REGION Network 7: ET01 >>> Lectura de CARA DELANTERA
   RUNG wire#powerrail
      Contact( #GAL_ET00 )
      Contact( #HabilitarLectura )
      Contact( #PermisoLectura )
      Contact( #pHsGalibo_OK )
      Contact( #pHs_LecturaDelantera_Des1 )
      Contact( #pHs_LecturaTrasera_Des1 )
      Contact( #pHs_LecturaDelantera_Des2 )
      Contact( #pHs_LecturaTrasera_Des2 )
      Contact( #pHs_LecturaDelantera_Error )
      Contact( #pHs_LecturaTrasera_Error )
      Contact( #EstadoZona.Marcha_CBx )
      I_Contact( #EstadoZona.Error_CBx )
      S_SR(operand := #GAL_ET01, r1 := wire#w1)
   END_RUNG
   RUNG wire#powerrail
      Contact( #GAL_ET02 )
   END_RUNG wire#w1
   RUNG wire#powerrail
      Contact( #EstadoZona.Resetear_CBx )
   END_RUNG wire#w1
   // the same network as SCL:
   IF #GAL_ET00 AND #HabilitarLectura AND #PermisoLectura AND #pHsGalibo_OK AND #pHs_LecturaDelantera_Des1 AND #pHs_LecturaTrasera_Des1 AND #pHs_LecturaDelantera_Des2 AND #pHs_LecturaTrasera_Des2 AND #pHs_LecturaDelantera_Error AND #pHs_LecturaTrasera_Error AND #EstadoZona.Marcha_CBx AND NOT #EstadoZona.Error_CBx THEN
       #GAL_ET01 := TRUE;   // SR flip-flop
   END_IF;
   IF #GAL_ET02 OR #EstadoZona.Resetear_CBx THEN #GAL_ET01 := FALSE; END_IF;
END_REGION

REGION Network 8: ET00 >>> INICIO
   RUNG wire#powerrail
      I_Contact( #GAL_ET00 )
      I_Contact( #GAL_ET01 )
      I_Contact( #GAL_ET02 )
      I_Contact( #GAL_ET03 )
      I_Contact( #GAL_ET04 )
      wire#w1
      S_SR(operand := #GAL_ET00, r1 := wire#w2)
   END_RUNG
   RUNG wire#powerrail
      Contact( #GAL_ET04 )
      I_Contact( #HabilitarLectura )
      I_Contact( #PermisoLectura )
      Contact( #pHsGalibo_OK )
      Contact( #pHs_LecturaDelantera_Des1 )
      Contact( #pHs_LecturaTrasera_Des1 )
      Contact( #pHs_LecturaDelantera_Des2 )
      Contact( #pHs_LecturaTrasera_Des2 )
      Contact( #pHs_LecturaDelantera_Error )
      Contact( #pHs_LecturaTrasera_Error )
   END_RUNG wire#w1
   RUNG wire#powerrail
      Contact( #GAL_ET01 )
   END_RUNG wire#w2
   RUNG wire#powerrail
      Contact( #EstadoZona.Resetear_CBx )
   END_RUNG wire#w2
   // the same network as SCL:
   IF (NOT #GAL_ET00 AND NOT #GAL_ET01 AND NOT #GAL_ET02 AND NOT #GAL_ET03 AND NOT #GAL_ET04) OR (#GAL_ET04 AND NOT #HabilitarLectura AND NOT #PermisoLectura AND #pHsGalibo_OK AND #pHs_LecturaDelantera_Des1 AND #pHs_LecturaTrasera_Des1 AND #pHs_LecturaDelantera_Des2 AND #pHs_LecturaTrasera_Des2 AND #pHs_LecturaDelantera_Error AND #pHs_LecturaTrasera_Error) THEN
       #GAL_ET00 := TRUE;   // SR flip-flop
   END_IF;
   IF #GAL_ET01 OR #EstadoZona.Resetear_CBx THEN #GAL_ET00 := FALSE; END_IF;
END_REGION

REGION Network 9: ERROR >>> Fotocelulas de Galibo
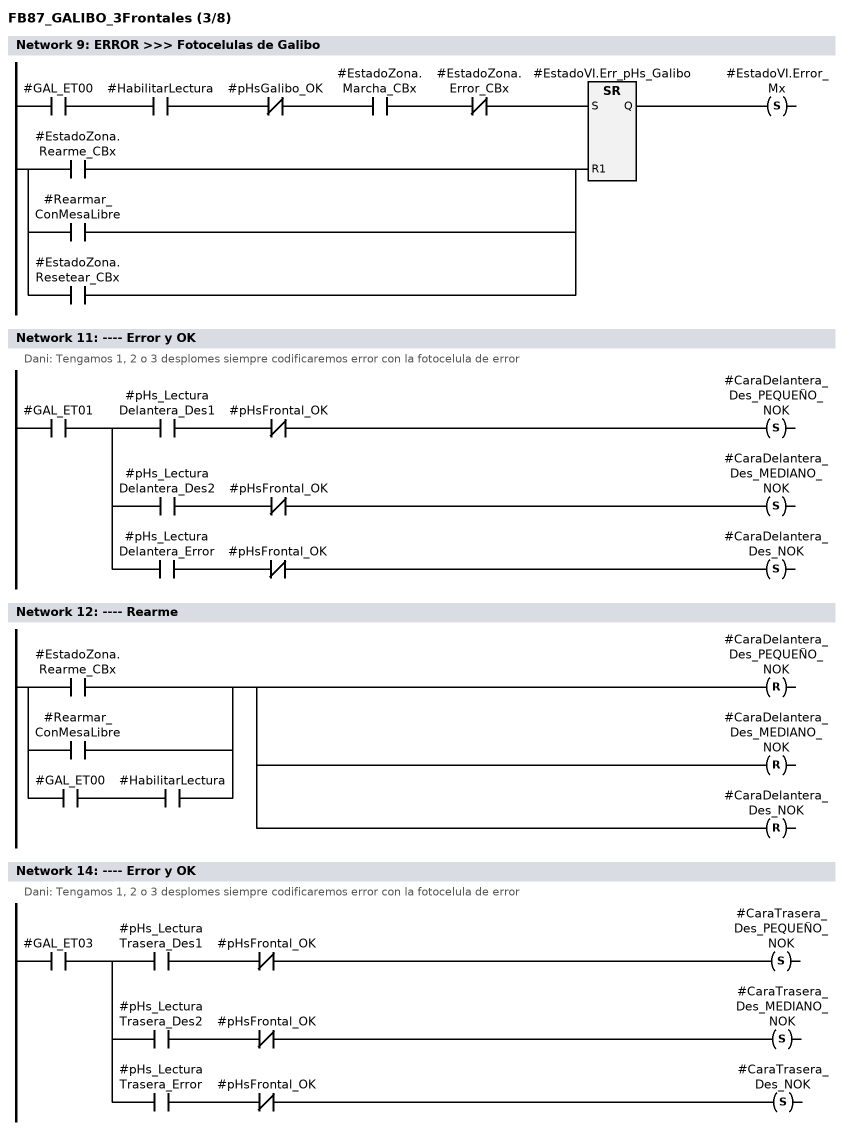
   RUNG wire#powerrail
      Contact( #GAL_ET00 )
      Contact( #HabilitarLectura )
      I_Contact( #pHsGalibo_OK )
      Contact( #EstadoZona.Marcha_CBx )
      I_Contact( #EstadoZona.Error_CBx )
      S_SR(operand := #EstadoVI.Err_pHs_Galibo, r1 := wire#w1)
      S_Coil( #EstadoVI.Error_Mx )
   END_RUNG
   RUNG wire#powerrail
      Contact( #EstadoZona.Rearme_CBx )
   END_RUNG wire#w1
   RUNG wire#powerrail
      Contact( #Rearmar_ConMesaLibre )
   END_RUNG wire#w1
   RUNG wire#powerrail
      Contact( #EstadoZona.Resetear_CBx )
   END_RUNG wire#w1
   // the same network as SCL:
   IF #GAL_ET00 AND #HabilitarLectura AND NOT #pHsGalibo_OK AND #EstadoZona.Marcha_CBx AND NOT #EstadoZona.Error_CBx THEN
       #EstadoVI.Err_pHs_Galibo := TRUE;   // SR flip-flop
   END_IF;
   IF #EstadoZona.Rearme_CBx OR #Rearmar_ConMesaLibre OR #EstadoZona.Resetear_CBx THEN
       #EstadoVI.Err_pHs_Galibo := FALSE;
   END_IF;
   IF #EstadoVI.Err_pHs_Galibo THEN #EstadoVI.Error_Mx := TRUE; END_IF;
END_REGION

REGION Network 10: VARIABLES DE CONTROL DE LARGURA >>> Activar la lectura de Cara Delantera
END_REGION

REGION Network 11: ---- Error y OK
   // Dani: Tengamos 1, 2 o 3 desplomes siempre codificaremos error con la fotocelula de error
   RUNG wire#powerrail
      Contact( #GAL_ET01 )
      wire#w1
      Contact( #pHs_LecturaDelantera_Des1 )
      I_Contact( #pHsFrontal_OK )
      S_Coil( #CaraDelantera_Des_PEQUEÑO_NOK )
   END_RUNG
   RUNG wire#w1
      Contact( #pHs_LecturaDelantera_Des2 )
      I_Contact( #pHsFrontal_OK )
      S_Coil( #CaraDelantera_Des_MEDIANO_NOK )
   END_RUNG
   RUNG wire#w1
      Contact( #pHs_LecturaDelantera_Error )
      I_Contact( #pHsFrontal_OK )
      S_Coil( #CaraDelantera_Des_NOK )
   END_RUNG
   // the same network as SCL:
   IF #GAL_ET01 AND #pHs_LecturaDelantera_Des1 AND NOT #pHsFrontal_OK THEN
       #CaraDelantera_Des_PEQUEÑO_NOK := TRUE;
   END_IF;
   IF #GAL_ET01 AND #pHs_LecturaDelantera_Des2 AND NOT #pHsFrontal_OK THEN
       #CaraDelantera_Des_MEDIANO_NOK := TRUE;
   END_IF;
   IF #GAL_ET01 AND #pHs_LecturaDelantera_Error AND NOT #pHsFrontal_OK THEN
       #CaraDelantera_Des_NOK := TRUE;
   END_IF;
END_REGION

REGION Network 12: ---- Rearme
   RUNG wire#powerrail
      Contact( #EstadoZona.Rearme_CBx )
      wire#w1
      R_Coil( #CaraDelantera_Des_PEQUEÑO_NOK )
   END_RUNG
   RUNG wire#powerrail
      Contact( #Rearmar_ConMesaLibre )
   END_RUNG wire#w1
   RUNG wire#powerrail
      Contact( #GAL_ET00 )
      Contact( #HabilitarLectura )
   END_RUNG wire#w1
   RUNG wire#w1
      R_Coil( #CaraDelantera_Des_MEDIANO_NOK )
   END_RUNG
   RUNG wire#w1
      R_Coil( #CaraDelantera_Des_NOK )
   END_RUNG
   // the same network as SCL:
   IF #EstadoZona.Rearme_CBx OR #Rearmar_ConMesaLibre OR (#GAL_ET00 AND #HabilitarLectura) THEN
       #CaraDelantera_Des_PEQUEÑO_NOK := FALSE;
       #CaraDelantera_Des_MEDIANO_NOK := FALSE;
       #CaraDelantera_Des_NOK := FALSE;
   END_IF;
END_REGION

REGION Network 13: VARIABLES DE CONTROL DE LARGURA >>> Activar la lectura de Cara Trasera
END_REGION

REGION Network 14: ---- Error y OK
   // Dani: Tengamos 1, 2 o 3 desplomes siempre codificaremos error con la fotocelula de error
   RUNG wire#powerrail
      Contact( #GAL_ET03 )
      wire#w1
      Contact( #pHs_LecturaTrasera_Des1 )
      I_Contact( #pHsFrontal_OK )
      S_Coil( #CaraTrasera_Des_PEQUEÑO_NOK )
   END_RUNG
   RUNG wire#w1
      Contact( #pHs_LecturaTrasera_Des2 )
      I_Contact( #pHsFrontal_OK )
      S_Coil( #CaraTrasera_Des_MEDIANO_NOK )
   END_RUNG
   RUNG wire#w1
      Contact( #pHs_LecturaTrasera_Error )
      I_Contact( #pHsFrontal_OK )
      S_Coil( #CaraTrasera_Des_NOK )
   END_RUNG
   // the same network as SCL:
   IF #GAL_ET03 AND #pHs_LecturaTrasera_Des1 AND NOT #pHsFrontal_OK THEN
       #CaraTrasera_Des_PEQUEÑO_NOK := TRUE;
   END_IF;
   IF #GAL_ET03 AND #pHs_LecturaTrasera_Des2 AND NOT #pHsFrontal_OK THEN
       #CaraTrasera_Des_MEDIANO_NOK := TRUE;
   END_IF;
   IF #GAL_ET03 AND #pHs_LecturaTrasera_Error AND NOT #pHsFrontal_OK THEN
       #CaraTrasera_Des_NOK := TRUE;
   END_IF;
END_REGION

REGION Network 15: ---- Rearme
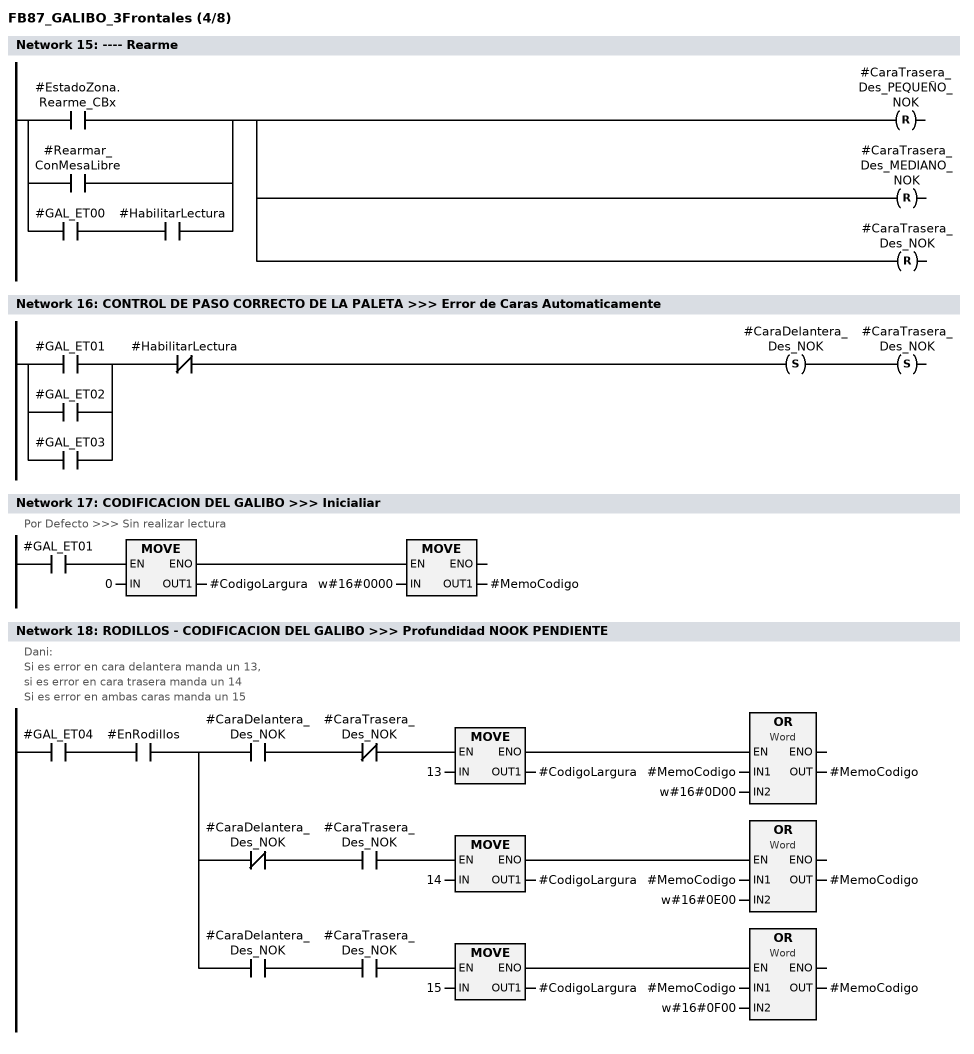
   RUNG wire#powerrail
      Contact( #EstadoZona.Rearme_CBx )
      wire#w1
      R_Coil( #CaraTrasera_Des_PEQUEÑO_NOK )
   END_RUNG
   RUNG wire#powerrail
      Contact( #Rearmar_ConMesaLibre )
   END_RUNG wire#w1
   RUNG wire#powerrail
      Contact( #GAL_ET00 )
      Contact( #HabilitarLectura )
   END_RUNG wire#w1
   RUNG wire#w1
      R_Coil( #CaraTrasera_Des_MEDIANO_NOK )
   END_RUNG
   RUNG wire#w1
      R_Coil( #CaraTrasera_Des_NOK )
   END_RUNG
   // the same network as SCL:
   IF #EstadoZona.Rearme_CBx OR #Rearmar_ConMesaLibre OR (#GAL_ET00 AND #HabilitarLectura) THEN
       #CaraTrasera_Des_PEQUEÑO_NOK := FALSE;
       #CaraTrasera_Des_MEDIANO_NOK := FALSE;
       #CaraTrasera_Des_NOK := FALSE;
   END_IF;
END_REGION

REGION Network 16: CONTROL DE PASO CORRECTO DE LA PALETA >>> Error de Caras Automaticamente
   RUNG wire#powerrail
      Contact( #GAL_ET01 )
      wire#w1
      I_Contact( #HabilitarLectura )
      S_Coil( #CaraDelantera_Des_NOK )
      S_Coil( #CaraTrasera_Des_NOK )
   END_RUNG
   RUNG wire#powerrail
      Contact( #GAL_ET02 )
   END_RUNG wire#w1
   RUNG wire#powerrail
      Contact( #GAL_ET03 )
   END_RUNG wire#w1
   // the same network as SCL:
   IF (#GAL_ET01 OR #GAL_ET02 OR #GAL_ET03) AND NOT #HabilitarLectura THEN
       #CaraDelantera_Des_NOK := TRUE;
       #CaraTrasera_Des_NOK := TRUE;
   END_IF;
END_REGION

REGION Network 17: CODIFICACION DEL GALIBO >>> Inicialiar
   // Por Defecto >>> Sin realizar lectura
   RUNG wire#powerrail
      Contact( #GAL_ET01 )
      { S7_GenerateENO := "TRUE" } Move(in := 0, out1 => #CodigoLargura)
      { S7_GenerateENO := "TRUE" } Move(in := w#16#0000, out1 => #MemoCodigo)
   END_RUNG
   // the same network as SCL:
   // ENO of a box is taken as its EN; it also drops when the box reports an error
   IF #GAL_ET01 THEN
       #CodigoLargura := 0;
       #MemoCodigo := w#16#0000;
   END_IF;
END_REGION

REGION Network 18: RODILLOS - CODIFICACION DEL GALIBO >>> Profundidad NOOK PENDIENTE
   // Dani:
   // Si es error en cara delantera manda un 13, 
   // si es error en cara trasera manda un 14
   // Si es error en ambas caras manda un 15
   #_w1 := #GAL_ET04 AND #EnRodillos;
   IF #_w1 AND #CaraDelantera_Des_NOK AND NOT #CaraTrasera_Des_NOK THEN
       #CodigoLargura := 13;
       #MemoCodigo := #MemoCodigo OR w#16#0D00;
   END_IF;
   IF #_w1 AND NOT #CaraDelantera_Des_NOK AND #CaraTrasera_Des_NOK THEN
       #CodigoLargura := 14;
       #MemoCodigo := #MemoCodigo OR w#16#0E00;
   END_IF;
   IF #_w1 AND #CaraDelantera_Des_NOK AND #CaraTrasera_Des_NOK THEN
       #CodigoLargura := 15;
       #MemoCodigo := #MemoCodigo OR w#16#0F00;
   END_IF;
END_REGION

REGION Network 19: RODILLOS - CODIFICACION DEL GALIBO >>> Profundidad OK - Codificacion
   // Dani:  los Nook solo se escriben si el desplome esta configurado
   // si hay 1 desplome envia 1 si la carga no da error de desplome
   // Si hay 2 desplomes envia 1 si no hay desplome pequeño y 2 si no hay error de desplome
   // Si hay 3 desplomes envia 1 si no hay desplome pequeño, 2 si no hay desplome mediano y 3 si no hay error de desplome
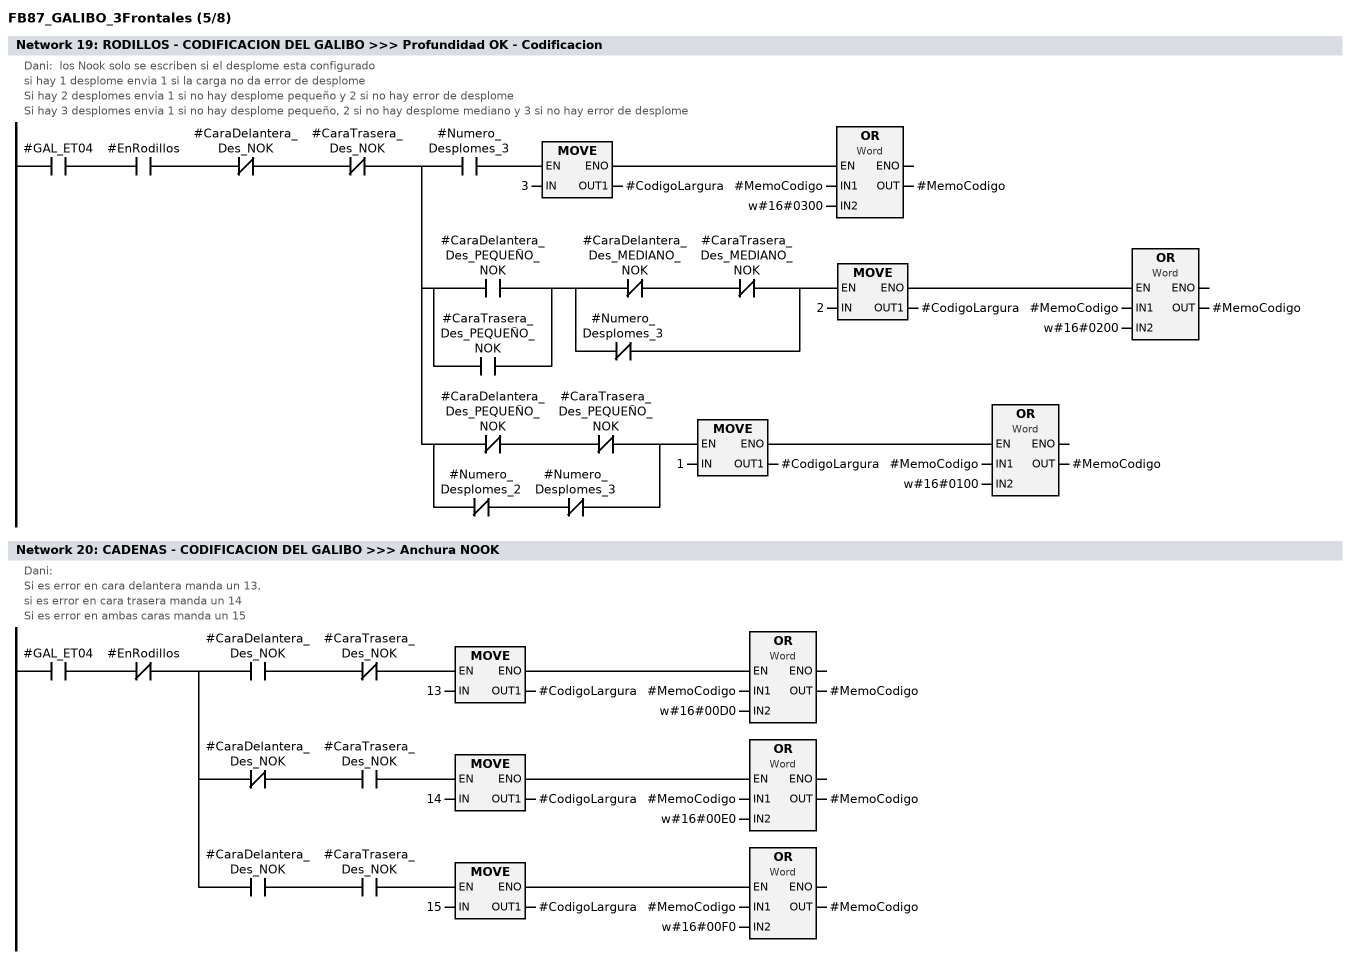
   #_w1 := #GAL_ET04 AND #EnRodillos AND NOT #CaraDelantera_Des_NOK AND NOT #CaraTrasera_Des_NOK;
   IF #_w1 AND #Numero_Desplomes_3 THEN
       #CodigoLargura := 3;
       #MemoCodigo := #MemoCodigo OR w#16#0300;
   END_IF;
   IF #_w1 AND (#CaraDelantera_Des_PEQUEÑO_NOK OR #CaraTrasera_Des_PEQUEÑO_NOK) AND ((NOT #CaraDelantera_Des_MEDIANO_NOK AND NOT #CaraTrasera_Des_MEDIANO_NOK) OR NOT #Numero_Desplomes_3) THEN
       #CodigoLargura := 2;
       #MemoCodigo := #MemoCodigo OR w#16#0200;
   END_IF;
   IF #_w1 AND ((NOT #CaraDelantera_Des_PEQUEÑO_NOK AND NOT #CaraTrasera_Des_PEQUEÑO_NOK) OR (NOT #Numero_Desplomes_2 AND NOT #Numero_Desplomes_3)) THEN
       #CodigoLargura := 1;
       #MemoCodigo := #MemoCodigo OR w#16#0100;
   END_IF;
END_REGION

REGION Network 20: CADENAS - CODIFICACION DEL GALIBO >>> Anchura NOOK
   // Dani:
   // Si es error en cara delantera manda un 13, 
   // si es error en cara trasera manda un 14
   // Si es error en ambas caras manda un 15
   #_w1 := #GAL_ET04 AND NOT #EnRodillos;
   IF #_w1 AND #CaraDelantera_Des_NOK AND NOT #CaraTrasera_Des_NOK THEN
       #CodigoLargura := 13;
       #MemoCodigo := #MemoCodigo OR w#16#00D0;
   END_IF;
   IF #_w1 AND NOT #CaraDelantera_Des_NOK AND #CaraTrasera_Des_NOK THEN
       #CodigoLargura := 14;
       #MemoCodigo := #MemoCodigo OR w#16#00E0;
   END_IF;
   IF #_w1 AND #CaraDelantera_Des_NOK AND #CaraTrasera_Des_NOK THEN
       #CodigoLargura := 15;
       #MemoCodigo := #MemoCodigo OR w#16#00F0;
   END_IF;
END_REGION

REGION Network 21: CADENAS - CODIFICACION DEL GALIBO >>> Anchura OK - Codificacion
   // Dani:
   // Si la cargaes menor que desplome 1 manda 1
   // si la carga es mayor que desplome 1 y menor que desplome 2 manda 2
   // si la carga es mayor que desplome 2 y menor que desplome 3 manda 3
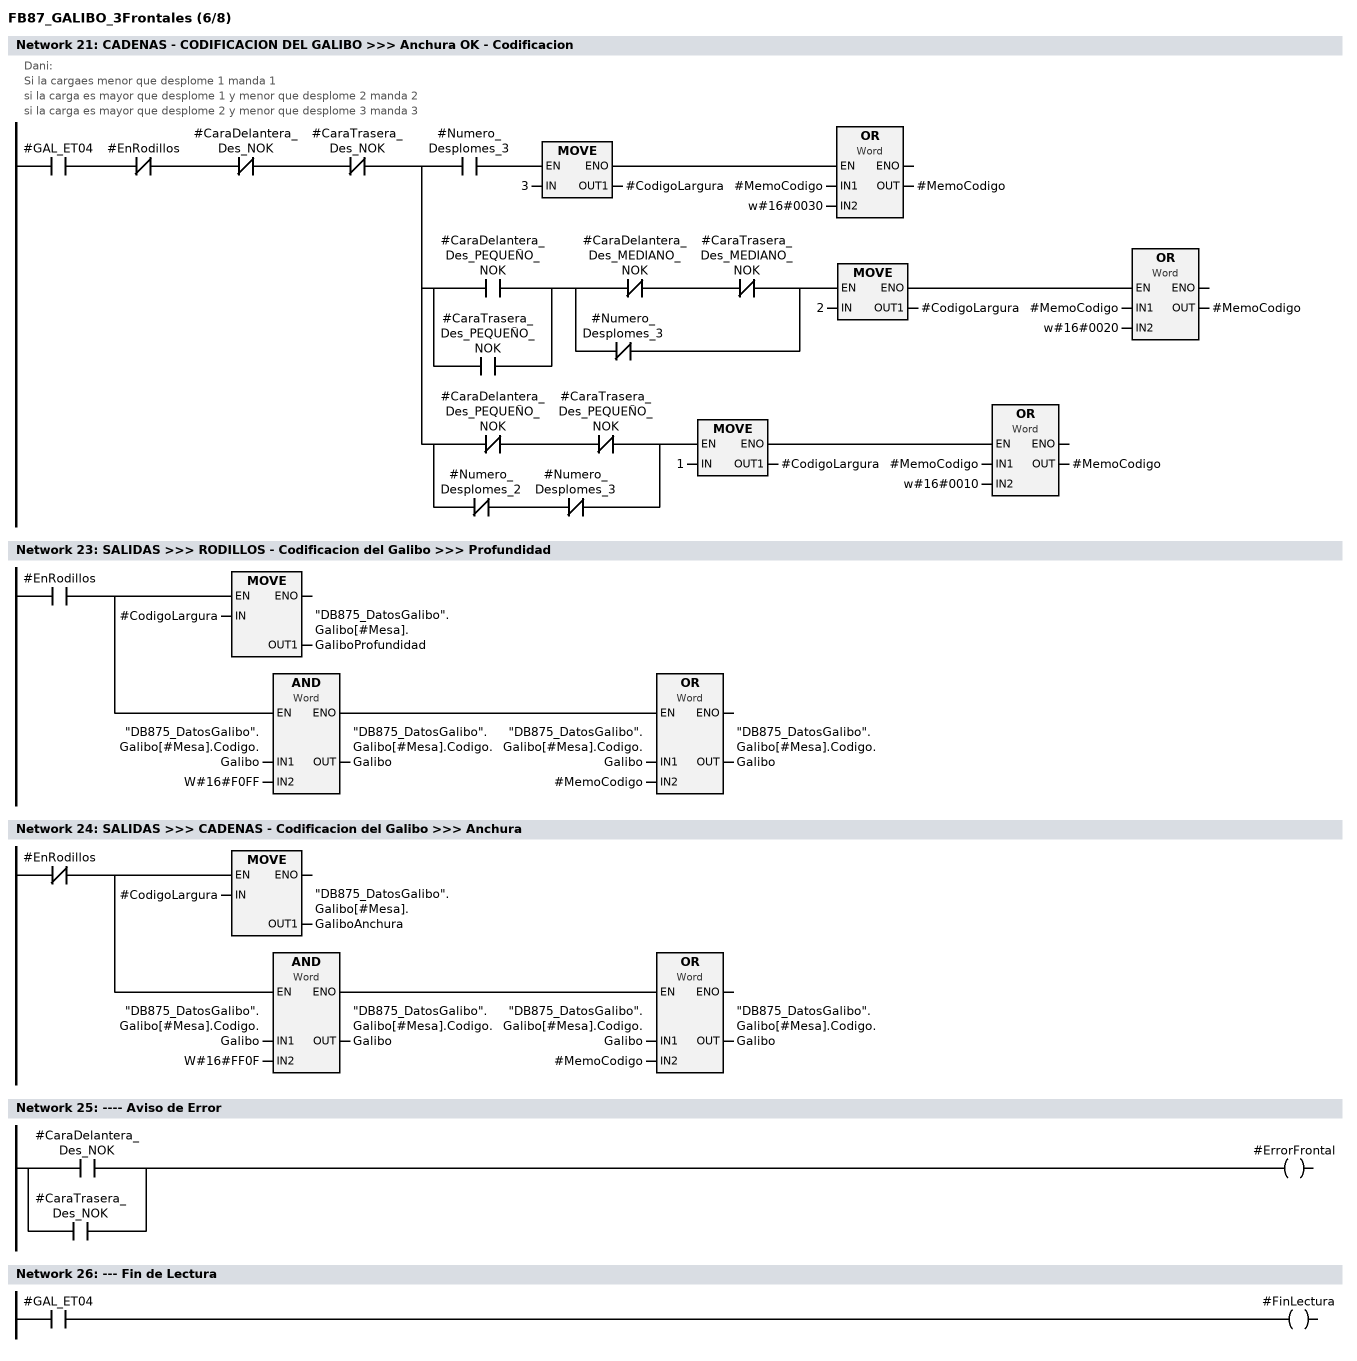
   #_w1 := #GAL_ET04 AND NOT #EnRodillos AND NOT #CaraDelantera_Des_NOK AND NOT #CaraTrasera_Des_NOK;
   IF #_w1 AND #Numero_Desplomes_3 THEN
       #CodigoLargura := 3;
       #MemoCodigo := #MemoCodigo OR w#16#0030;
   END_IF;
   IF #_w1 AND (#CaraDelantera_Des_PEQUEÑO_NOK OR #CaraTrasera_Des_PEQUEÑO_NOK) AND ((NOT #CaraDelantera_Des_MEDIANO_NOK AND NOT #CaraTrasera_Des_MEDIANO_NOK) OR NOT #Numero_Desplomes_3) THEN
       #CodigoLargura := 2;
       #MemoCodigo := #MemoCodigo OR w#16#0020;
   END_IF;
   IF #_w1 AND ((NOT #CaraDelantera_Des_PEQUEÑO_NOK AND NOT #CaraTrasera_Des_PEQUEÑO_NOK) OR (NOT #Numero_Desplomes_2 AND NOT #Numero_Desplomes_3)) THEN
       #CodigoLargura := 1;
       #MemoCodigo := #MemoCodigo OR w#16#0010;
   END_IF;
END_REGION

REGION Network 22: SALIDAS >>> Codificacion del Galibo y Error de Anchura
END_REGION

REGION Network 23: SALIDAS >>> RODILLOS - Codificacion del Galibo >>> Profundidad
   IF #EnRodillos THEN
       "DB875_DatosGalibo".Galibo[#Mesa].GaliboProfundidad := #CodigoLargura;
       "DB875_DatosGalibo".Galibo[#Mesa].Codigo.Galibo := "DB875_DatosGalibo".Galibo[#Mesa].Codigo.Galibo AND W#16#F0FF;
       "DB875_DatosGalibo".Galibo[#Mesa].Codigo.Galibo := "DB875_DatosGalibo".Galibo[#Mesa].Codigo.Galibo OR #MemoCodigo;
   END_IF;
END_REGION

REGION Network 24: SALIDAS >>> CADENAS - Codificacion del Galibo >>> Anchura
   IF NOT #EnRodillos THEN
       "DB875_DatosGalibo".Galibo[#Mesa].GaliboAnchura := #CodigoLargura;
       "DB875_DatosGalibo".Galibo[#Mesa].Codigo.Galibo := "DB875_DatosGalibo".Galibo[#Mesa].Codigo.Galibo AND W#16#FF0F;
       "DB875_DatosGalibo".Galibo[#Mesa].Codigo.Galibo := "DB875_DatosGalibo".Galibo[#Mesa].Codigo.Galibo OR #MemoCodigo;
   END_IF;
END_REGION

REGION Network 25: ---- Aviso de Error
   RUNG wire#powerrail
      Contact( #CaraDelantera_Des_NOK )
      wire#w1
      Coil( #ErrorFrontal )
   END_RUNG
   RUNG wire#powerrail
      Contact( #CaraTrasera_Des_NOK )
   END_RUNG wire#w1
   // the same network as SCL:
   #ErrorFrontal := #CaraDelantera_Des_NOK OR #CaraTrasera_Des_NOK;
END_REGION

REGION Network 26: --- Fin de Lectura
   RUNG wire#powerrail
      Contact( #GAL_ET04 )
      Coil( #FinLectura )
   END_RUNG
   // the same network as SCL:
   #FinLectura := #GAL_ET04;
END_REGION

REGION Network 27: SALIDAS >>> BALIZA
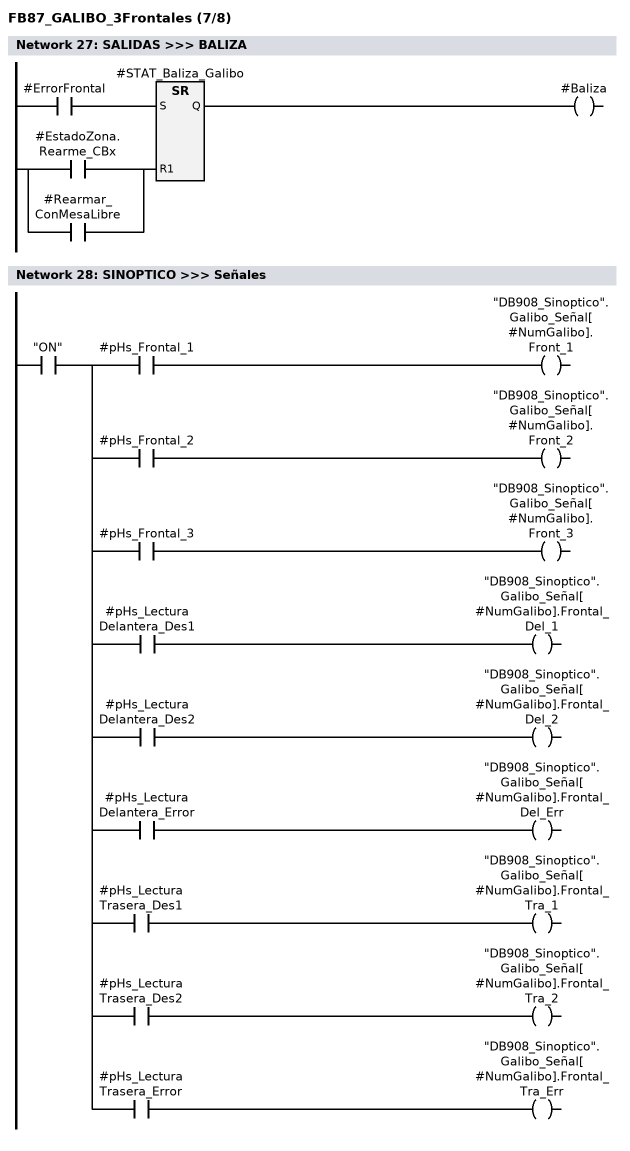
   RUNG wire#powerrail
      Contact( #ErrorFrontal )
      S_SR(operand := #STAT_Baliza_Galibo, r1 := wire#w1)
      Coil( #Baliza )
   END_RUNG
   RUNG wire#powerrail
      Contact( #EstadoZona.Rearme_CBx )
   END_RUNG wire#w1
   RUNG wire#powerrail
      Contact( #Rearmar_ConMesaLibre )
   END_RUNG wire#w1
   // the same network as SCL:
   IF #ErrorFrontal THEN
       #STAT_Baliza_Galibo := TRUE;   // SR flip-flop
   END_IF;
   IF #EstadoZona.Rearme_CBx OR #Rearmar_ConMesaLibre THEN #STAT_Baliza_Galibo := FALSE; END_IF;
   #Baliza := #STAT_Baliza_Galibo;
END_REGION

REGION Network 28: SINOPTICO >>> Señales
   RUNG wire#powerrail
      Contact( "ON" )
      wire#w1
      Contact( #pHs_Frontal_1 )
      Coil( "DB908_Sinoptico".Galibo_Señal[#NumGalibo].Front_1 )
   END_RUNG
   RUNG wire#w1
      Contact( #pHs_Frontal_2 )
      Coil( "DB908_Sinoptico".Galibo_Señal[#NumGalibo].Front_2 )
   END_RUNG
   RUNG wire#w1
      Contact( #pHs_Frontal_3 )
      Coil( "DB908_Sinoptico".Galibo_Señal[#NumGalibo].Front_3 )
   END_RUNG
   RUNG wire#w1
      Contact( #pHs_LecturaDelantera_Des1 )
      Coil( "DB908_Sinoptico".Galibo_Señal[#NumGalibo].Frontal_Del_1 )
   END_RUNG
   RUNG wire#w1
      Contact( #pHs_LecturaDelantera_Des2 )
      Coil( "DB908_Sinoptico".Galibo_Señal[#NumGalibo].Frontal_Del_2 )
   END_RUNG
   RUNG wire#w1
      Contact( #pHs_LecturaDelantera_Error )
      Coil( "DB908_Sinoptico".Galibo_Señal[#NumGalibo].Frontal_Del_Err )
   END_RUNG
   RUNG wire#w1
      Contact( #pHs_LecturaTrasera_Des1 )
      Coil( "DB908_Sinoptico".Galibo_Señal[#NumGalibo].Frontal_Tra_1 )
   END_RUNG
   RUNG wire#w1
      Contact( #pHs_LecturaTrasera_Des2 )
      Coil( "DB908_Sinoptico".Galibo_Señal[#NumGalibo].Frontal_Tra_2 )
   END_RUNG
   RUNG wire#w1
      Contact( #pHs_LecturaTrasera_Error )
      Coil( "DB908_Sinoptico".Galibo_Señal[#NumGalibo].Frontal_Tra_Err )
   END_RUNG
   // the same network as SCL:
   "DB908_Sinoptico".Galibo_Señal[#NumGalibo].Front_1 := "ON" AND #pHs_Frontal_1;
   "DB908_Sinoptico".Galibo_Señal[#NumGalibo].Front_2 := "ON" AND #pHs_Frontal_2;
   "DB908_Sinoptico".Galibo_Señal[#NumGalibo].Front_3 := "ON" AND #pHs_Frontal_3;
   "DB908_Sinoptico".Galibo_Señal[#NumGalibo].Frontal_Del_1 := "ON" AND #pHs_LecturaDelantera_Des1;
   "DB908_Sinoptico".Galibo_Señal[#NumGalibo].Frontal_Del_2 := "ON" AND #pHs_LecturaDelantera_Des2;
   "DB908_Sinoptico".Galibo_Señal[#NumGalibo].Frontal_Del_Err := "ON" AND #pHs_LecturaDelantera_Error;
   "DB908_Sinoptico".Galibo_Señal[#NumGalibo].Frontal_Tra_1 := "ON" AND #pHs_LecturaTrasera_Des1;
   "DB908_Sinoptico".Galibo_Señal[#NumGalibo].Frontal_Tra_2 := "ON" AND #pHs_LecturaTrasera_Des2;
   "DB908_Sinoptico".Galibo_Señal[#NumGalibo].Frontal_Tra_Err := "ON" AND #pHs_LecturaTrasera_Error;
END_REGION

REGION Network 29: SINOPTICO >>> RODILLOS >>> Codigo >>> Profundidad
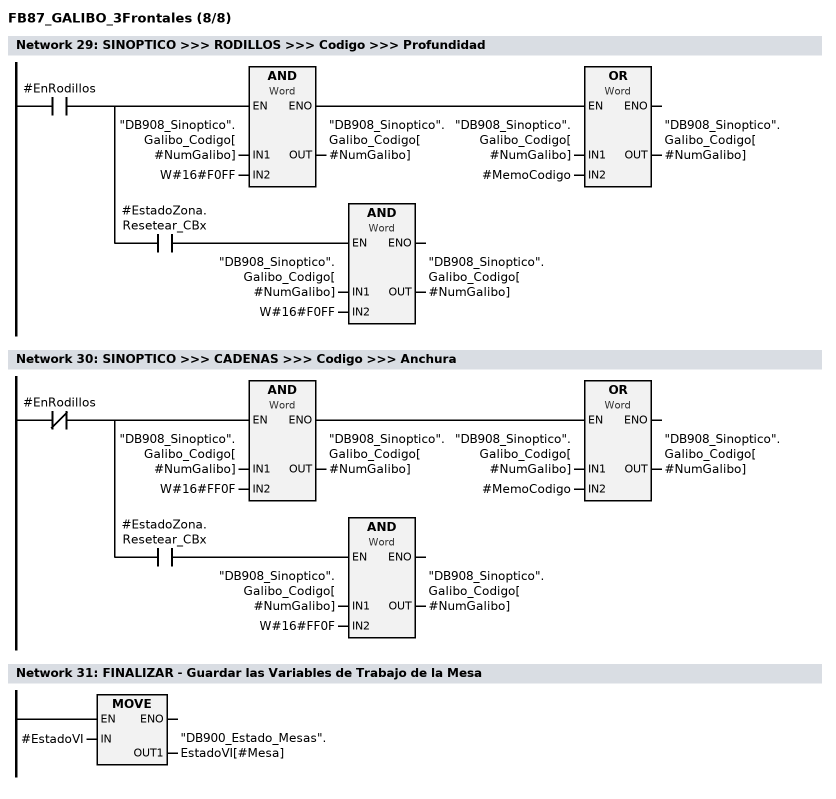
   IF #EnRodillos THEN
       "DB908_Sinoptico".Galibo_Codigo[#NumGalibo] := "DB908_Sinoptico".Galibo_Codigo[#NumGalibo] AND W#16#F0FF;
       "DB908_Sinoptico".Galibo_Codigo[#NumGalibo] := "DB908_Sinoptico".Galibo_Codigo[#NumGalibo] OR #MemoCodigo;
   END_IF;
   IF #EnRodillos AND #EstadoZona.Resetear_CBx THEN
       "DB908_Sinoptico".Galibo_Codigo[#NumGalibo] := "DB908_Sinoptico".Galibo_Codigo[#NumGalibo] AND W#16#F0FF;
   END_IF;
END_REGION

REGION Network 30: SINOPTICO >>> CADENAS >>> Codigo >>> Anchura
   IF NOT #EnRodillos THEN
       "DB908_Sinoptico".Galibo_Codigo[#NumGalibo] := "DB908_Sinoptico".Galibo_Codigo[#NumGalibo] AND W#16#FF0F;
       "DB908_Sinoptico".Galibo_Codigo[#NumGalibo] := "DB908_Sinoptico".Galibo_Codigo[#NumGalibo] OR #MemoCodigo;
   END_IF;
   IF NOT #EnRodillos AND #EstadoZona.Resetear_CBx THEN
       "DB908_Sinoptico".Galibo_Codigo[#NumGalibo] := "DB908_Sinoptico".Galibo_Codigo[#NumGalibo] AND W#16#FF0F;
   END_IF;
END_REGION

REGION Network 31: FINALIZAR - Guardar las Variables de Trabajo de la Mesa
   RUNG wire#powerrail
      Move(in := #EstadoVI, out1 => "DB900_Estado_Mesas".EstadoVI[#Mesa])
   END_RUNG
   // the same network as SCL:
   "DB900_Estado_Mesas".EstadoVI[#Mesa] := #EstadoVI;
END_REGION
END_FUNCTION_BLOCK

FUNCTION_BLOCK "FB89_GALIBO_Remontada_EnRodillos"   // FB89, LAD
TITLE = Galibo de 5 Alturas (2023)
{ S7_Optimized_Access := 'FALSE' }
AUTHOR : GALIBO
NAME : 20140101
VERSION : 3.0
// stored: AutoNumber false, SetENOAutomatically false
   VAR_INPUT
      Mesa : UInt;
      NumGalibo : UInt;
      pHs_Remontado_1Dcha : Bool;
      pHs_Remontado_2Dcha : Bool;
      pHs_Remontado_1Izq : Bool;
      pHs_Remontado_2Izq : Bool;
      HabilitarLectura : Bool;
      PermisoLectura : Bool;
      Rearmar_ConMesaLibre : Bool;
      V_Estabilidad : Int;
   END_VAR
   VAR_OUTPUT
      Codigo : Word;
      FinLectura : Bool;
   END_VAR
   VAR_IN_OUT
      SinopticoGalibo_Señal : "UDT_HMI_SeñalesGalibo";
      SinopticoGalibo_Codigo : Word;
   END_VAR
   VAR
      CNT_Estabilidad : "FB910_CNT_UHS";
      GAL_ET00 : Bool;
      GAL_ET01 : Bool;
      GAL_ET02 : Bool;
      GAL_ET03 : Bool;
      pHsGalibo_OK { ExternalAccessible := 'False'; ExternalVisible := 'False'; ExternalWritable := 'False'} : Bool;
      LeerRemontado : Bool;
      FinRemontado : Bool;
      Remontado_NO : Bool;
      Remontado_SI : Bool;
      CodigoRemontado : SInt;
      MemoCodigo : Word;
      STAT_Baliza_Galibo : Bool;
   END_VAR
   VAR_TEMP
      EstadoZona : "EstadoZona";
      EstadoVI : "EstadosMesa";
   END_VAR
BEGIN

REGION Network 1: INICIALIZAR - Recoger las Variables de Estado de la Mesa
   // Se recoge - Estado_CBx
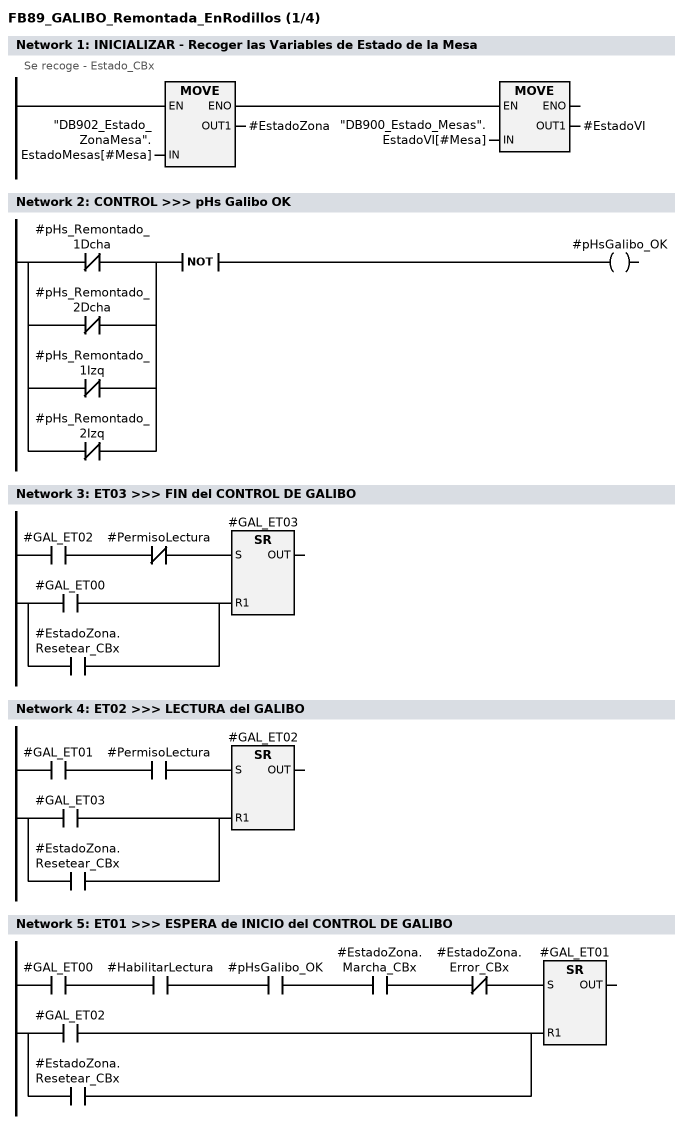
   RUNG wire#powerrail
      Move(in := "DB902_Estado_ZonaMesa".EstadoMesas[#Mesa], out1 => #EstadoZona)
      Move(in := "DB900_Estado_Mesas".EstadoVI[#Mesa], out1 => #EstadoVI)
   END_RUNG
   // the same network as SCL:
   #EstadoZona := "DB902_Estado_ZonaMesa".EstadoMesas[#Mesa];
   #EstadoVI := "DB900_Estado_Mesas".EstadoVI[#Mesa];
END_REGION

REGION Network 2: CONTROL >>> pHs Galibo OK
   RUNG wire#powerrail
      I_Contact( #pHs_Remontado_1Dcha )
      wire#w1
      Not()
      Coil( #pHsGalibo_OK )
   END_RUNG
   RUNG wire#powerrail
      I_Contact( #pHs_Remontado_2Dcha )
   END_RUNG wire#w1
   RUNG wire#powerrail
      I_Contact( #pHs_Remontado_1Izq )
   END_RUNG wire#w1
   RUNG wire#powerrail
      I_Contact( #pHs_Remontado_2Izq )
   END_RUNG wire#w1
   // the same network as SCL:
   #pHsGalibo_OK := NOT (NOT #pHs_Remontado_1Dcha OR NOT #pHs_Remontado_2Dcha OR NOT #pHs_Remontado_1Izq OR NOT #pHs_Remontado_2Izq);
END_REGION

REGION Network 3: ET03 >>> FIN del CONTROL DE GALIBO
   RUNG wire#powerrail
      Contact( #GAL_ET02 )
      I_Contact( #PermisoLectura )
      S_SR(operand := #GAL_ET03, r1 := wire#w1)
   END_RUNG
   RUNG wire#powerrail
      Contact( #GAL_ET00 )
   END_RUNG wire#w1
   RUNG wire#powerrail
      Contact( #EstadoZona.Resetear_CBx )
   END_RUNG wire#w1
   // the same network as SCL:
   IF #GAL_ET02 AND NOT #PermisoLectura THEN
       #GAL_ET03 := TRUE;   // SR flip-flop
   END_IF;
   IF #GAL_ET00 OR #EstadoZona.Resetear_CBx THEN #GAL_ET03 := FALSE; END_IF;
END_REGION

REGION Network 4: ET02 >>> LECTURA del GALIBO
   RUNG wire#powerrail
      Contact( #GAL_ET01 )
      Contact( #PermisoLectura )
      S_SR(operand := #GAL_ET02, r1 := wire#w1)
   END_RUNG
   RUNG wire#powerrail
      Contact( #GAL_ET03 )
   END_RUNG wire#w1
   RUNG wire#powerrail
      Contact( #EstadoZona.Resetear_CBx )
   END_RUNG wire#w1
   // the same network as SCL:
   IF #GAL_ET01 AND #PermisoLectura THEN
       #GAL_ET02 := TRUE;   // SR flip-flop
   END_IF;
   IF #GAL_ET03 OR #EstadoZona.Resetear_CBx THEN #GAL_ET02 := FALSE; END_IF;
END_REGION

REGION Network 5: ET01 >>> ESPERA de INICIO del CONTROL DE GALIBO
   RUNG wire#powerrail
      Contact( #GAL_ET00 )
      Contact( #HabilitarLectura )
      Contact( #pHsGalibo_OK )
      Contact( #EstadoZona.Marcha_CBx )
      I_Contact( #EstadoZona.Error_CBx )
      S_SR(operand := #GAL_ET01, r1 := wire#w1)
   END_RUNG
   RUNG wire#powerrail
      Contact( #GAL_ET02 )
   END_RUNG wire#w1
   RUNG wire#powerrail
      Contact( #EstadoZona.Resetear_CBx )
   END_RUNG wire#w1
   // the same network as SCL:
   IF #GAL_ET00 AND #HabilitarLectura AND #pHsGalibo_OK AND #EstadoZona.Marcha_CBx AND NOT #EstadoZona.Error_CBx THEN
       #GAL_ET01 := TRUE;   // SR flip-flop
   END_IF;
   IF #GAL_ET02 OR #EstadoZona.Resetear_CBx THEN #GAL_ET01 := FALSE; END_IF;
END_REGION

REGION Network 6: ET00 >>> INICIO
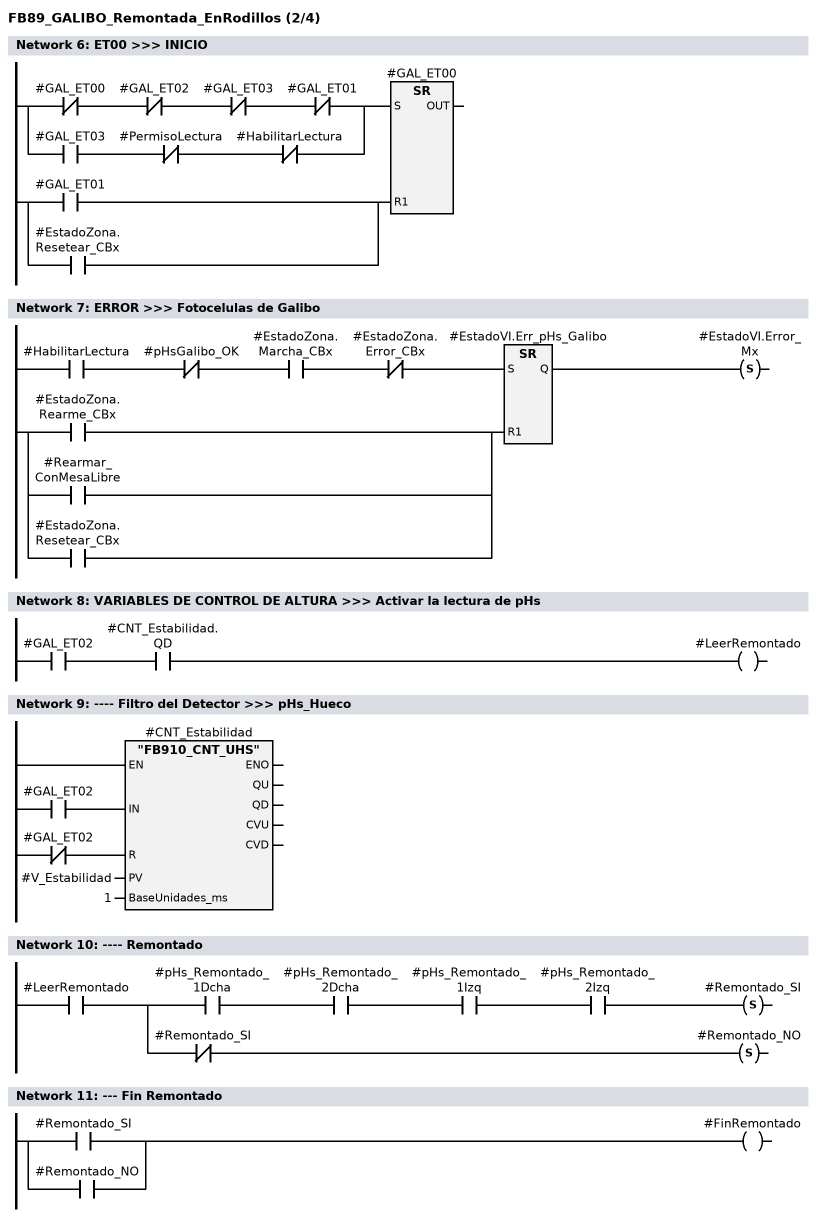
   RUNG wire#powerrail
      I_Contact( #GAL_ET00 )
      I_Contact( #GAL_ET02 )
      I_Contact( #GAL_ET03 )
      I_Contact( #GAL_ET01 )
      wire#w1
      S_SR(operand := #GAL_ET00, r1 := wire#w2)
   END_RUNG
   RUNG wire#powerrail
      Contact( #GAL_ET03 )
      I_Contact( #PermisoLectura )
      I_Contact( #HabilitarLectura )
   END_RUNG wire#w1
   RUNG wire#powerrail
      Contact( #GAL_ET01 )
   END_RUNG wire#w2
   RUNG wire#powerrail
      Contact( #EstadoZona.Resetear_CBx )
   END_RUNG wire#w2
   // the same network as SCL:
   IF (NOT #GAL_ET00 AND NOT #GAL_ET02 AND NOT #GAL_ET03 AND NOT #GAL_ET01) OR (#GAL_ET03 AND NOT #PermisoLectura AND NOT #HabilitarLectura) THEN
       #GAL_ET00 := TRUE;   // SR flip-flop
   END_IF;
   IF #GAL_ET01 OR #EstadoZona.Resetear_CBx THEN #GAL_ET00 := FALSE; END_IF;
END_REGION

REGION Network 7: ERROR >>> Fotocelulas de Galibo
   RUNG wire#powerrail
      Contact( #HabilitarLectura )
      I_Contact( #pHsGalibo_OK )
      Contact( #EstadoZona.Marcha_CBx )
      I_Contact( #EstadoZona.Error_CBx )
      S_SR(operand := #EstadoVI.Err_pHs_Galibo, r1 := wire#w1)
      S_Coil( #EstadoVI.Error_Mx )
   END_RUNG
   RUNG wire#powerrail
      Contact( #EstadoZona.Rearme_CBx )
   END_RUNG wire#w1
   RUNG wire#powerrail
      Contact( #Rearmar_ConMesaLibre )
   END_RUNG wire#w1
   RUNG wire#powerrail
      Contact( #EstadoZona.Resetear_CBx )
   END_RUNG wire#w1
   // the same network as SCL:
   IF #HabilitarLectura AND NOT #pHsGalibo_OK AND #EstadoZona.Marcha_CBx AND NOT #EstadoZona.Error_CBx THEN
       #EstadoVI.Err_pHs_Galibo := TRUE;   // SR flip-flop
   END_IF;
   IF #EstadoZona.Rearme_CBx OR #Rearmar_ConMesaLibre OR #EstadoZona.Resetear_CBx THEN
       #EstadoVI.Err_pHs_Galibo := FALSE;
   END_IF;
   IF #EstadoVI.Err_pHs_Galibo THEN #EstadoVI.Error_Mx := TRUE; END_IF;
END_REGION

REGION Network 8: VARIABLES DE CONTROL DE ALTURA >>> Activar la lectura de pHs
   RUNG wire#powerrail
      Contact( #GAL_ET02 )
      Contact( #CNT_Estabilidad.QD )
      Coil( #LeerRemontado )
   END_RUNG
   // the same network as SCL:
   #LeerRemontado := #GAL_ET02 AND #CNT_Estabilidad.QD;
END_REGION

REGION Network 9: ---- Filtro del Detector >>> pHs_Hueco
   RUNG wire#powerrail
      #CNT_Estabilidad(IN := wire#w1, R := wire#w2, PV := #V_Estabilidad, BaseUnidades_ms := 1, QU =>, QD =>, CVU =>, CVD =>)
   END_RUNG
   RUNG wire#powerrail
      Contact( #GAL_ET02 )
   END_RUNG wire#w1
   RUNG wire#powerrail
      I_Contact( #GAL_ET02 )
   END_RUNG wire#w2
   // the same network as SCL:
   #CNT_Estabilidad(IN := #GAL_ET02, R := NOT #GAL_ET02, PV := #V_Estabilidad, BaseUnidades_ms := 1);   // "FB910_CNT_UHS"
END_REGION

REGION Network 10: ---- Remontado
   RUNG wire#powerrail
      Contact( #LeerRemontado )
      wire#w1
      Contact( #pHs_Remontado_1Dcha )
      Contact( #pHs_Remontado_2Dcha )
      Contact( #pHs_Remontado_1Izq )
      Contact( #pHs_Remontado_2Izq )
      S_Coil( #Remontado_SI )
   END_RUNG
   RUNG wire#w1
      I_Contact( #Remontado_SI )
      S_Coil( #Remontado_NO )
   END_RUNG
   // the same network as SCL:
   IF #LeerRemontado AND #pHs_Remontado_1Dcha AND #pHs_Remontado_2Dcha AND #pHs_Remontado_1Izq AND #pHs_Remontado_2Izq THEN
       #Remontado_SI := TRUE;
   END_IF;
   IF #LeerRemontado AND NOT #Remontado_SI THEN #Remontado_NO := TRUE; END_IF;
END_REGION

REGION Network 11: --- Fin Remontado
   RUNG wire#powerrail
      Contact( #Remontado_SI )
      wire#w1
      Coil( #FinRemontado )
   END_RUNG
   RUNG wire#powerrail
      Contact( #Remontado_NO )
   END_RUNG wire#w1
   // the same network as SCL:
   #FinRemontado := #Remontado_SI OR #Remontado_NO;
END_REGION

REGION Network 12: --- Rearme
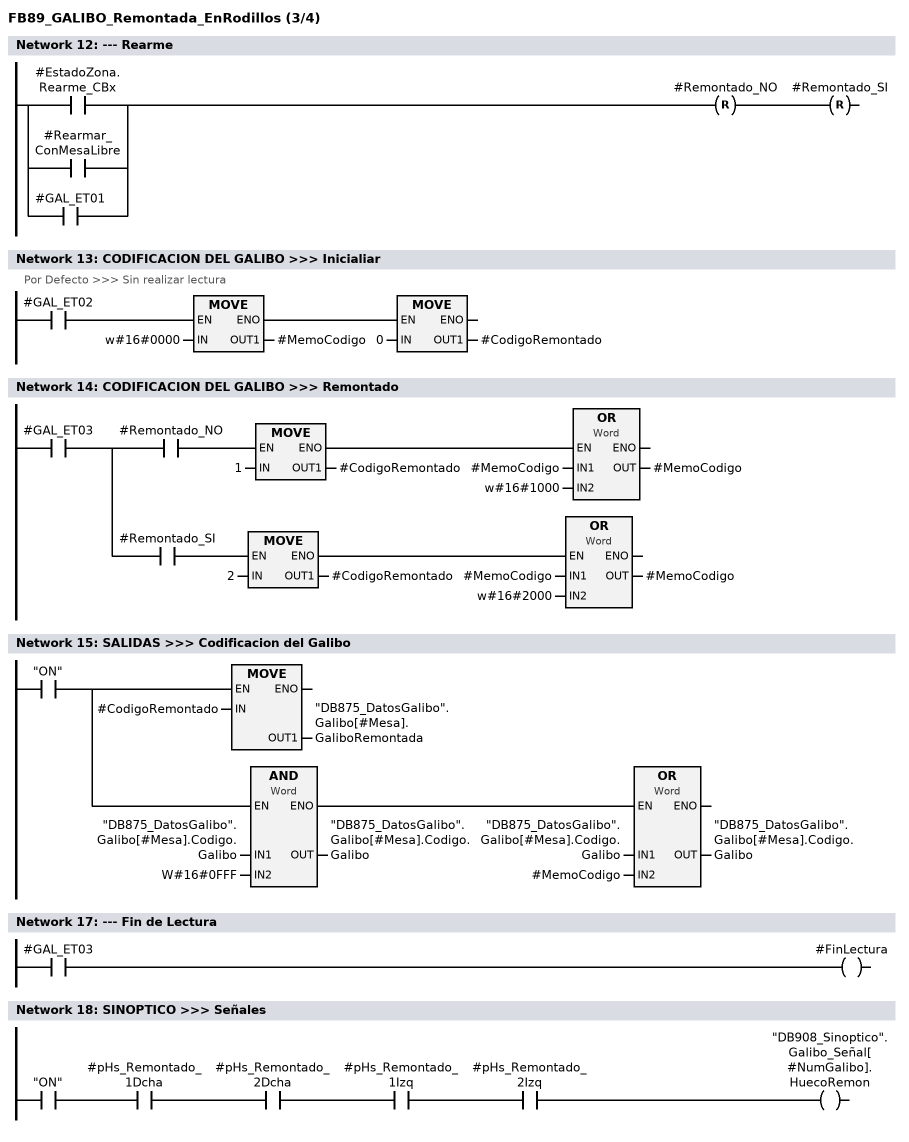
   RUNG wire#powerrail
      Contact( #EstadoZona.Rearme_CBx )
      wire#w1
      R_Coil( #Remontado_NO )
      R_Coil( #Remontado_SI )
   END_RUNG
   RUNG wire#powerrail
      Contact( #Rearmar_ConMesaLibre )
   END_RUNG wire#w1
   RUNG wire#powerrail
      Contact( #GAL_ET01 )
   END_RUNG wire#w1
   // the same network as SCL:
   IF #EstadoZona.Rearme_CBx OR #Rearmar_ConMesaLibre OR #GAL_ET01 THEN
       #Remontado_NO := FALSE;
       #Remontado_SI := FALSE;
   END_IF;
END_REGION

REGION Network 13: CODIFICACION DEL GALIBO >>> Inicialiar
   // Por Defecto >>> Sin realizar lectura
   RUNG wire#powerrail
      Contact( #GAL_ET02 )
      { S7_GenerateENO := "TRUE" } Move(in := w#16#0000, out1 => #MemoCodigo)
      { S7_GenerateENO := "TRUE" } Move(in := 0, out1 => #CodigoRemontado)
   END_RUNG
   // the same network as SCL:
   // ENO of a box is taken as its EN; it also drops when the box reports an error
   IF #GAL_ET02 THEN
       #MemoCodigo := w#16#0000;
       #CodigoRemontado := 0;
   END_IF;
END_REGION

REGION Network 14: CODIFICACION DEL GALIBO >>> Remontado
   // ENO of a box is taken as its EN; it also drops when the box reports an error
   IF #GAL_ET03 AND #Remontado_NO THEN
       #CodigoRemontado := 1;
       #MemoCodigo := #MemoCodigo OR w#16#1000;
   END_IF;
   IF #GAL_ET03 AND #Remontado_SI THEN
       #CodigoRemontado := 2;
       #MemoCodigo := #MemoCodigo OR w#16#2000;
   END_IF;
END_REGION

REGION Network 15: SALIDAS >>> Codificacion del Galibo
   IF "ON" THEN
       "DB875_DatosGalibo".Galibo[#Mesa].GaliboRemontada := #CodigoRemontado;
       "DB875_DatosGalibo".Galibo[#Mesa].Codigo.Galibo := "DB875_DatosGalibo".Galibo[#Mesa].Codigo.Galibo AND W#16#0FFF;
       "DB875_DatosGalibo".Galibo[#Mesa].Codigo.Galibo := "DB875_DatosGalibo".Galibo[#Mesa].Codigo.Galibo OR #MemoCodigo;
   END_IF;
END_REGION

REGION Network 16: ---- Aviso de Error NOTA >>> NO PROCEDE
END_REGION

REGION Network 17: --- Fin de Lectura
   RUNG wire#powerrail
      Contact( #GAL_ET03 )
      Coil( #FinLectura )
   END_RUNG
   // the same network as SCL:
   #FinLectura := #GAL_ET03;
END_REGION

REGION Network 18: SINOPTICO >>> Señales
   RUNG wire#powerrail
      Contact( "ON" )
      Contact( #pHs_Remontado_1Dcha )
      Contact( #pHs_Remontado_2Dcha )
      Contact( #pHs_Remontado_1Izq )
      Contact( #pHs_Remontado_2Izq )
      Coil( "DB908_Sinoptico".Galibo_Señal[#NumGalibo].HuecoRemon )
   END_RUNG
   // the same network as SCL:
   "DB908_Sinoptico".Galibo_Señal[#NumGalibo].HuecoRemon := "ON" AND #pHs_Remontado_1Dcha AND #pHs_Remontado_2Dcha AND #pHs_Remontado_1Izq AND #pHs_Remontado_2Izq;
END_REGION

REGION Network 19: SINOPTICO >>> Codigo
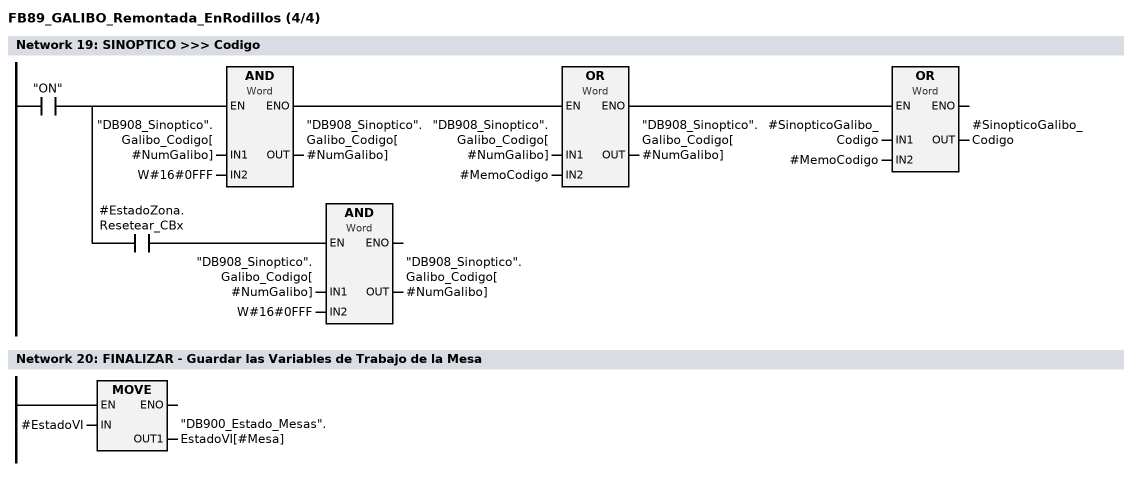
   IF "ON" THEN
       "DB908_Sinoptico".Galibo_Codigo[#NumGalibo] := "DB908_Sinoptico".Galibo_Codigo[#NumGalibo] AND W#16#0FFF;
       "DB908_Sinoptico".Galibo_Codigo[#NumGalibo] := "DB908_Sinoptico".Galibo_Codigo[#NumGalibo] OR #MemoCodigo;
       #SinopticoGalibo_Codigo := #SinopticoGalibo_Codigo OR #MemoCodigo;
   END_IF;
   IF "ON" AND #EstadoZona.Resetear_CBx THEN
       "DB908_Sinoptico".Galibo_Codigo[#NumGalibo] := "DB908_Sinoptico".Galibo_Codigo[#NumGalibo] AND W#16#0FFF;
   END_IF;
END_REGION

REGION Network 20: FINALIZAR - Guardar las Variables de Trabajo de la Mesa
   RUNG wire#powerrail
      Move(in := #EstadoVI, out1 => "DB900_Estado_Mesas".EstadoVI[#Mesa])
   END_RUNG
   // the same network as SCL:
   "DB900_Estado_Mesas".EstadoVI[#Mesa] := #EstadoVI;
END_REGION
END_FUNCTION_BLOCK

FUNCTION_BLOCK "FB830_PasarDatosEntrePLCs_Origen"   // FB830, LAD
{ S7_Optimized_Access := 'FALSE' }
// stored: AutoNumber false, SetENOAutomatically false
   VAR_INPUT
      Mesa : UInt;
      OrdenEvacuar : Bool;
      In_BorrarUT : Bool;
   END_VAR
   VAR_OUTPUT
      Out_Mckey_01 : "UDT_EntrePLCs";
      Out_McKey_02 : "UDT_EntrePLCs";
      Out_DatosUT : Bool;
      OrdenEvacuar_OK : Bool;
   END_VAR
   VAR
      MMckeyUT_01 : "UDT_EntrePLCs";
      MMcKeyUT_02 : "UDT_EntrePLCs";
      NumeroUT_01 { ExternalAccessible := 'False'; ExternalVisible := 'False'; ExternalWritable := 'False'} : UInt;
      NumeroUT_02 { ExternalAccessible := 'False'; ExternalVisible := 'False'; ExternalWritable := 'False'} : UInt;
      ExisteUT_01 : Bool;
      ExisteUT_02 : Bool;
      MFP_BorrarUT : Bool;
      MDatosUT : Bool;
      MOrdenOK : Bool;
   END_VAR
   VAR_TEMP
      EstadoZona : "EstadoZona";
      EstadoVI : "EstadosMesa";
      Mckey_01 : "UDT_EntrePLCs";
      Mckey_02 : "UDT_EntrePLCs";
      P_Temporal : DWord;
      ValorReturn : Int;
      Cero : Byte;
      OrdenBorrarUT : Bool;
   END_VAR
   VAR_TEMP   // added for the SCL form of the ladder/FBD networks
      _w1 : Bool;
      _w2 : Bool;
      _w3 : Bool;
   END_VAR
BEGIN

REGION Network 1: Inicializar Variables
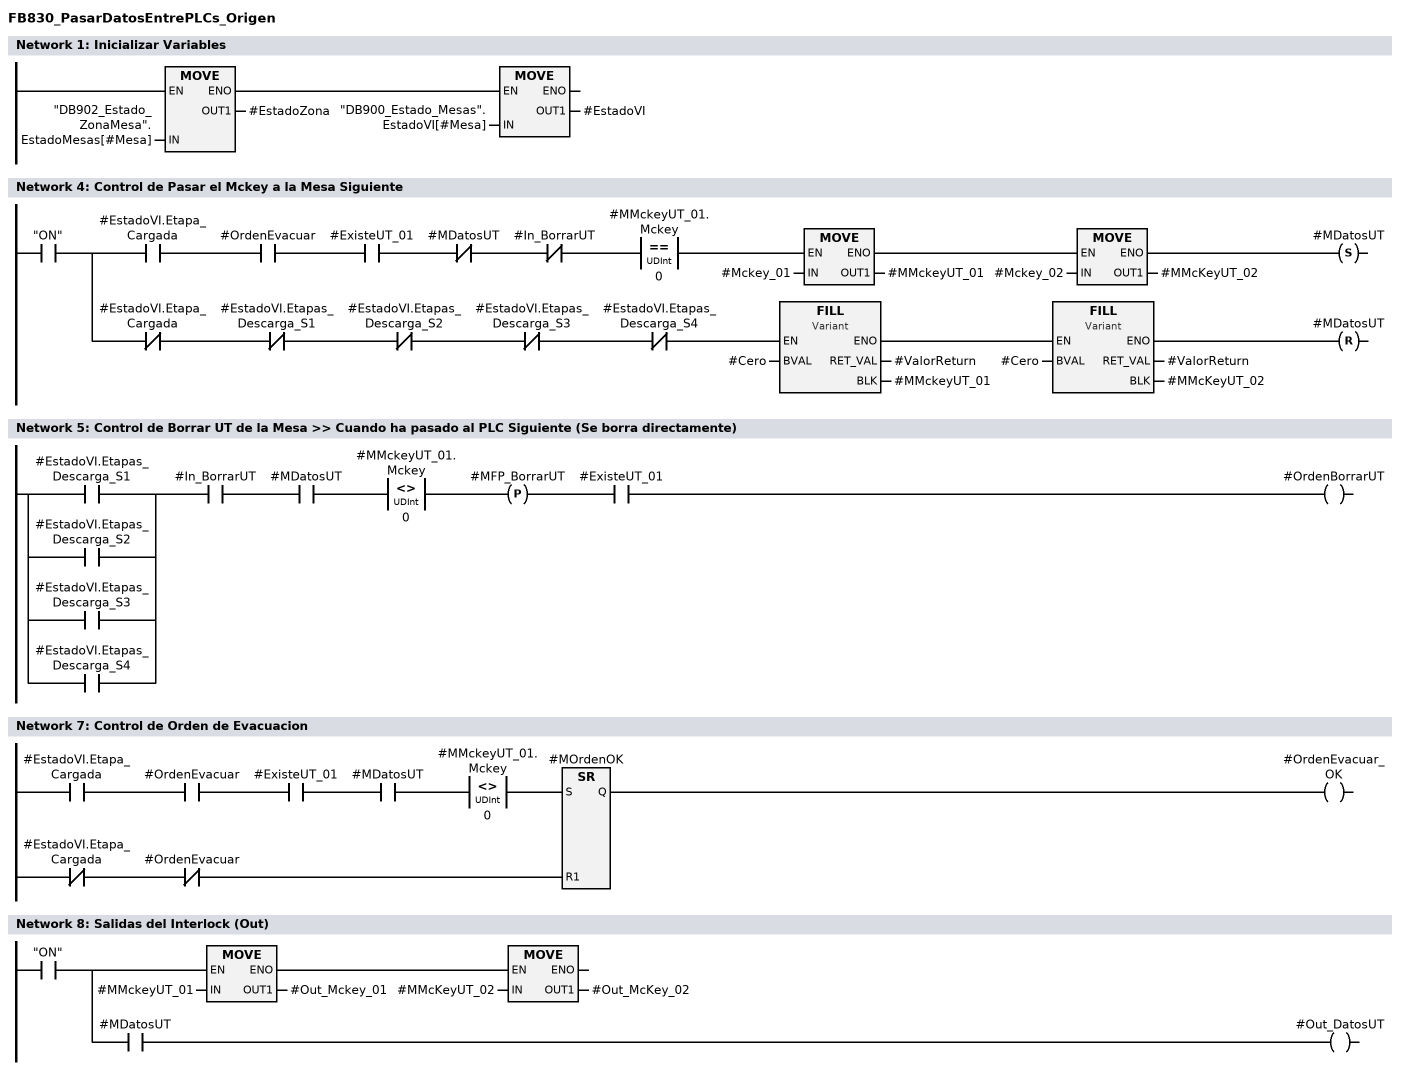
   RUNG wire#powerrail
      Move(in := "DB902_Estado_ZonaMesa".EstadoMesas[#Mesa], out1 => #EstadoZona)
      Move(in := "DB900_Estado_Mesas".EstadoVI[#Mesa], out1 => #EstadoVI)
   END_RUNG
   // the same network as SCL:
   #EstadoZona := "DB902_Estado_ZonaMesa".EstadoMesas[#Mesa];
   #EstadoVI := "DB900_Estado_Mesas".EstadoVI[#Mesa];
END_REGION

NETWORK
TITLE = ---
/////////////////////////////////////////////////////////////////////////////////
/////////////////////////////////////////////////////////////////////////////////
/////////////////////////////////////////////////////////////////////////////////
/// --- Inicializar Variables
      L     0;
      T     #Cero;


NETWORK
TITLE = Obtener Datos UT en la Mesa Actual
/////////////////////////////////////////////////////////////////////////////////
/////////////////////////////////////////////////////////////////////////////////
/////////////////////////////////////////////////////////////////////////////////
/// --- Inicializar

      SET;  // Inicializacion
      R     #ExisteUT_01;  // No Existe UT
      R     #ExisteUT_02;

      L     0;
      T     #NumeroUT_01;
      T     #NumeroUT_02;

      CALL  FILL
      ( BVAL    := #Cero,
        RET_VAL := #ValorReturn,
        BLK     := #Mckey_01
      );
      CALL  FILL
      ( BVAL    := #Cero,
        RET_VAL := #ValorReturn,
        BLK     := #Mckey_02
      );


/////////////////////////////////////////////////////////////////////////////////
/// --- Buscar Primera UT de la Mesa

      L     "DB810_ColasMesas".Colas[#Mesa].UT_PrimeraMesa;
      T     #NumeroUT_01;

      L     #NumeroUT_01;  // No hay UT's ?
      L     0;
      ==I;
      JC    FinDatosUTs_EnMesa;


/////////////////////////////////////////////////////////////////////////////////
/////////////////////////////////////////////////////////////////////////////////
/////////////////////////////////////////////////////////////////////////////////
/// --- Existe UT en la Mesa >>> Recoger Datos
      SET;
      S     #ExisteUT_01;  // Existe UT

      L     "DB812_UTs_Control".UT[#NumeroUT_01].Mckey;
      T     #Mckey_01.Mckey;
      L     "DB812_UTs_Control".UT[#NumeroUT_01].Grupo;
      T     #Mckey_01.Grupo;
      L     "DB812_UTs_Control".UT[#NumeroUT_01].TipoCarga;
      T     #Mckey_01.TipoCarga;

      L     "DB812_UTs_Control".UT[#NumeroUT_01].MesaDestino;
      T     #Mckey_01.MesaDestino;
      L     "DB813_UTs_Ruta".UT[#NumeroUT_01].Ruta[0];
      T     #Mckey_01.MesaSiguienteRuta;

      SET;
      A     "DB812_UTs_Control".UT[#NumeroUT_01].AtributosDelaCarga.Vacia;
      =     #Mckey_01.AtributosDelaCarga.Vacia;
      SET;
      A     "DB812_UTs_Control".UT[#NumeroUT_01].AtributosDelaCarga.Pila;
      =     #Mckey_01.AtributosDelaCarga.Pila;
      SET;
      A     "DB812_UTs_Control".UT[#NumeroUT_01].AtributosDelaCarga.Remontada;
      =     #Mckey_01.AtributosDelaCarga.Remontada;


/////////////////////////////////////////////////////////////////////////////////
/// --- Comprobar si puede haber mas

      L     "DB812_UTs_Control".UT[#NumeroUT_01].Grupo;
      L     0;  // Si es Grupo = 0 No hay mas
      ==I;
      JC    FinDatosUTs_EnMesa;

      L     "DB812_UTs_Control".UT[#NumeroUT_01].UT_SiguienteMesa;  // Hay mas UTs en la Mesa
      L     0;
      ==I;
      JC    FinDatosUTs_EnMesa;


/////////////////////////////////////////////////////////////////////////////////
/////////////////////////////////////////////////////////////////////////////////
/////////////////////////////////////////////////////////////////////////////////
/// --- Recoger datos de la Segunda UT

      L     "DB812_UTs_Control".UT[#NumeroUT_01].UT_SiguienteMesa;
      T     #NumeroUT_02;  // Puntero a los Datos de la UT

      SET;
      S     #ExisteUT_02;  // Existe UT

      L     "DB812_UTs_Control".UT[#NumeroUT_02].Mckey;
      T     #Mckey_02.Mckey;
      L     "DB812_UTs_Control".UT[#NumeroUT_02].Grupo;
      T     #Mckey_02.Grupo;
      L     "DB812_UTs_Control".UT[#NumeroUT_02].TipoCarga;
      T     #Mckey_02.TipoCarga;

      L     "DB812_UTs_Control".UT[#NumeroUT_02].MesaDestino;
      T     #Mckey_02.MesaDestino;
      L     "DB813_UTs_Ruta".UT[#NumeroUT_02].Ruta[0];
      T     #Mckey_02.MesaSiguienteRuta;

      SET;
      A     "DB812_UTs_Control".UT[#NumeroUT_02].AtributosDelaCarga.Vacia;
      =     #Mckey_02.AtributosDelaCarga.Vacia;
      SET;
      A     "DB812_UTs_Control".UT[#NumeroUT_02].AtributosDelaCarga.Pila;
      =     #Mckey_02.AtributosDelaCarga.Pila;
      SET;
      A     "DB812_UTs_Control".UT[#NumeroUT_02].AtributosDelaCarga.Remontada;
      =     #Mckey_02.AtributosDelaCarga.Remontada;


/////////////////////////////////////////////////////////////////////////////////
/// --- Comprobar si son pareja

      L     "DB812_UTs_Control".UT[#NumeroUT_01].Grupo;  // Son el mismo Grupo
      L     "DB812_UTs_Control".UT[#NumeroUT_02].Grupo;
      ==I;
      JC    FinDatosUTs_EnMesa;


/////////////////////////////////////////////////////////////////////////////////
/// --- Borrado de Datos no son el mismo grupo

      SET;
      R     #ExisteUT_02;

      L     0;
      T     #NumeroUT_02;

      CALL  FILL
      ( BVAL    := #Cero,
        RET_VAL := #ValorReturn,
        BLK     := #Mckey_01
      );


/////////////////////////////////////////////////////////////////////////////////
/////////////////////////////////////////////////////////////////////////////////
/////////////////////////////////////////////////////////////////////////////////
/// --- Final de Lectura de Datos de la UT en La Mesa
FinDatosUTs_EnMesa:NOP   0;



REGION Network 4: Control de Pasar el Mckey a la Mesa Siguiente
   RUNG wire#powerrail
      Contact( "ON" )
      wire#w1
      Contact( #EstadoVI.Etapa_Cargada )
      Contact( #OrdenEvacuar )
      Contact( #ExisteUT_01 )
      I_Contact( #MDatosUT )
      I_Contact( #In_BorrarUT )
      { S7_Templates := "SrcType := UDInt" } EQ_Contact(in1 := #MMckeyUT_01.Mckey, in2 := 0)
      { S7_GenerateENO := "TRUE" } Move(in := #Mckey_01, out1 => #MMckeyUT_01)
      { S7_GenerateENO := "TRUE" } Move(in := #Mckey_02, out1 => #MMcKeyUT_02)
      S_Coil( #MDatosUT )
   END_RUNG
   RUNG wire#w1
      I_Contact( #EstadoVI.Etapa_Cargada )
      I_Contact( #EstadoVI.Etapas_Descarga_S1 )
      I_Contact( #EstadoVI.Etapas_Descarga_S2 )
      I_Contact( #EstadoVI.Etapas_Descarga_S3 )
      I_Contact( #EstadoVI.Etapas_Descarga_S4 )
      { S7_Templates := "ptr_type := Variant" } FILL(BVAL := #Cero, RET_VAL => #ValorReturn, BLK => #MMckeyUT_01)
      { S7_Templates := "ptr_type := Variant" } FILL(BVAL := #Cero, RET_VAL => #ValorReturn, BLK => #MMcKeyUT_02)
      R_Coil( #MDatosUT )
   END_RUNG
   // the same network as SCL:
   // ENO of a box is taken as its EN; it also drops when the box reports an error
   #_w1 := "ON" AND #EstadoVI.Etapa_Cargada AND #OrdenEvacuar AND #ExisteUT_01 AND NOT #MDatosUT AND NOT #In_BorrarUT AND (#MMckeyUT_01.Mckey = 0);
   IF #_w1 THEN
       #MMckeyUT_01 := #Mckey_01;
       #MMcKeyUT_02 := #Mckey_02;
       #MDatosUT := TRUE;
   END_IF;
   #ValorReturn := FILL(EN := "ON" AND NOT #EstadoVI.Etapa_Cargada AND NOT #EstadoVI.Etapas_Descarga_S1 AND NOT #EstadoVI.Etapas_Descarga_S2 AND NOT #EstadoVI.Etapas_Descarga_S3 AND NOT #EstadoVI.Etapas_Descarga_S4,
                        BVAL := #Cero,
                        BLK => #MMckeyUT_01,
                        ENO => #_w2);
   #ValorReturn := FILL(EN := #_w2, BVAL := #Cero, BLK => #MMcKeyUT_02, ENO => #_w3);
   IF #_w3 THEN #MDatosUT := FALSE; END_IF;
END_REGION

REGION Network 5: Control de Borrar UT de la Mesa >> Cuando ha pasado al PLC Siguiente (Se borra directamente)
   RUNG wire#powerrail
      Contact( #EstadoVI.Etapas_Descarga_S1 )
      wire#w1
      Contact( #In_BorrarUT )
      Contact( #MDatosUT )
      { S7_Templates := "SrcType := UDInt" } NE_Contact(in1 := #MMckeyUT_01.Mckey, in2 := 0)
      P_Trig( #MFP_BorrarUT )
      Contact( #ExisteUT_01 )
      Coil( #OrdenBorrarUT )
   END_RUNG
   RUNG wire#powerrail
      Contact( #EstadoVI.Etapas_Descarga_S2 )
   END_RUNG wire#w1
   RUNG wire#powerrail
      Contact( #EstadoVI.Etapas_Descarga_S3 )
   END_RUNG wire#w1
   RUNG wire#powerrail
      Contact( #EstadoVI.Etapas_Descarga_S4 )
   END_RUNG wire#w1
   // the same network as SCL:
   #_w1 := (#EstadoVI.Etapas_Descarga_S1 OR #EstadoVI.Etapas_Descarga_S2 OR #EstadoVI.Etapas_Descarga_S3 OR #EstadoVI.Etapas_Descarga_S4) AND #In_BorrarUT AND #MDatosUT AND (#MMckeyUT_01.Mckey <> 0);
   #_w2 := #_w1 AND NOT #MFP_BorrarUT;   // rising edge
   #MFP_BorrarUT := #_w1;
   #OrdenBorrarUT := #_w2 AND #ExisteUT_01;
END_REGION

NETWORK
TITLE = --
/////////////////////////////////////////////////////////////////////////////////
/////////////////////////////////////////////////////////////////////////////////
/////////////////////////////////////////////////////////////////////////////////
/// - Ordem de Borrar

      SET;  // Hay que BorrarUT
      AN    #OrdenBorrarUT;
      JC    FinBorrarUT_EnMesa;


/////////////////////////////////////////////////////////////////////////////////
/////////////////////////////////////////////////////////////////////////////////
/////////////////////////////////////////////////////////////////////////////////
      SET;  // Eliminar datos Memorizados
      R     #MDatosUT;

      CALL  FILL
      ( BVAL    := #Cero,
        RET_VAL := #ValorReturn,
        BLK     := #MMckeyUT_01
      );
      CALL  FILL
      ( BVAL    := #Cero,
        RET_VAL := #ValorReturn,
        BLK     := #MMcKeyUT_02
      );


/////////////////////////////////////////////////////////////////////////////////
      SET;
      AN    #ExisteUT_01;  // Existe UT 01 en la Mesa
      JC    FinBorrarUT_EnMesa;

      CALL  "FC722_EliminarUT_DeMesa"
      ( NumeroUT := #NumeroUT_01
      );  //Eliminar la Primera UT de la mesa


      AN    #ExisteUT_02;  // Existe UT 02 en la Mesa
      JC    FinBorrarUT_EnMesa;

      CALL  "FC722_EliminarUT_DeMesa"
      ( NumeroUT := #NumeroUT_02
      );  //Eliminar la Segunda UT de la mesa


/////////////////////////////////////////////////////////////////////////////////
/////////////////////////////////////////////////////////////////////////////////
/////////////////////////////////////////////////////////////////////////////////
FinBorrarUT_EnMesa:NOP   0;



REGION Network 7: Control de Orden de Evacuacion
   RUNG wire#powerrail
      Contact( #EstadoVI.Etapa_Cargada )
      Contact( #OrdenEvacuar )
      Contact( #ExisteUT_01 )
      Contact( #MDatosUT )
      { S7_Templates := "SrcType := UDInt" } NE_Contact(in1 := #MMckeyUT_01.Mckey, in2 := 0)
      S_SR(operand := #MOrdenOK, r1 := wire#w1)
      Coil( #OrdenEvacuar_OK )
   END_RUNG
   RUNG wire#powerrail
      I_Contact( #EstadoVI.Etapa_Cargada )
      I_Contact( #OrdenEvacuar )
   END_RUNG wire#w1
   // the same network as SCL:
   IF #EstadoVI.Etapa_Cargada AND #OrdenEvacuar AND #ExisteUT_01 AND #MDatosUT AND (#MMckeyUT_01.Mckey <> 0) THEN
       #MOrdenOK := TRUE;   // SR flip-flop
   END_IF;
   IF NOT #EstadoVI.Etapa_Cargada AND NOT #OrdenEvacuar THEN #MOrdenOK := FALSE; END_IF;
   #OrdenEvacuar_OK := #MOrdenOK;
END_REGION

REGION Network 8: Salidas del Interlock (Out)
   RUNG wire#powerrail
      Contact( "ON" )
      wire#w1
      Move(in := #MMckeyUT_01, out1 => #Out_Mckey_01)
      Move(in := #MMcKeyUT_02, out1 => #Out_McKey_02)
   END_RUNG
   RUNG wire#w1
      Contact( #MDatosUT )
      Coil( #Out_DatosUT )
   END_RUNG
   // the same network as SCL:
   IF "ON" THEN
       #Out_Mckey_01 := #MMckeyUT_01;
       #Out_McKey_02 := #MMcKeyUT_02;
   END_IF;
   #Out_DatosUT := "ON" AND #MDatosUT;
END_REGION
END_FUNCTION_BLOCK

FUNCTION_BLOCK "FB989_Envio Datos Movimot Asi"   // FB989, SCL
{ S7_Optimized_Access := 'FALSE' }
VERSION : 0.0
// Parámetros del bloque
// stored: AutoNumber false, SetENOAutomatically false
   VAR_INPUT
      Dir_GW_ASI_Com : Int;   // Direccion de inicio de Command Interface del Gateway ASI de Bihl+Wiedemann
      Num_Line : Int;
      Num_Slave : Int;
      Valor_V1 : Real;   // Porcentaje de velocidad respecto de la maxima en formato REAL
      Valor_V2 : Real;
      Valor_V3 : Real;
      Valor_V4 : Real;
      Valor_V5 : Real;
      Valor_V6 : Real;
      Valor_V7 : Real;
      Valor_Rampa : Int;   // Rampa de aceleración en milisegundos
      Escritura : Bool;
      Solo_Velocidades : Bool;
      Solo_Rampa : Bool;
   END_VAR
   VAR_OUTPUT
      Finalizado : Bool;
      Con_Error : Bool;
   END_VAR
   VAR
      Lista_ComVel : Array[1..33] of Byte;
      Lista_ComRampa : Array[1..8] of Byte;
      Escritura_OLD : Bool;
      Ciclo_envio : Int;
   END_VAR
   VAR_TEMP
      Valor_W : Int;
      Valor_B AT Valor_W : Struct
         high : Byte;
         low : Byte;
      END_STRUCT;
      Flanco_Escritura : Bool;
      i : Int;
   END_VAR
BEGIN


       // Área de instrucciones
       #Flanco_Escritura := #Escritura AND NOT #Escritura_OLD ;


       IF #Flanco_Escritura THEN

           //cabecera envio Velocidades
           #Lista_ComVel[1] := 16#7D ;
           #Lista_ComVel[2] := INT_TO_BYTE (#Num_Line - 1);
           #Lista_ComVel[3] := 16#0A ;
           #Lista_ComVel[4] := INT_TO_BYTE (#Num_Slave);  //Num Esclavo ASI
           #Lista_ComVel[5] := 16#0A ;
           //velocidades (nos deben meter un porcentaje, y nosotros ajustar para que el 100.0% sea 16#4000, que en decimal es 16384, y /100=163.84)
           (* classic code: #Valor_W := REAL_TO_INT (#Valor_V1 * 163.84) ;*)
           #Valor_W := REAL_TO_INT (#Valor_V1 * REAL#163.84) ;
           #Lista_ComVel[6] := #Valor_B.high ;
           #Lista_ComVel[7] := #Valor_B.low ;
           #Valor_W := #Valor_W * (-1);
           #Lista_ComVel[8] := #Valor_B.high ;
           #Lista_ComVel[9] := #Valor_B.low ;
           (* classic code: #Valor_W := REAL_TO_INT (#Valor_V2 * 163.84) ;*)
           #Valor_W := REAL_TO_INT (#Valor_V2 * REAL#163.84) ;
           #Lista_ComVel[10] := #Valor_B.high ;
           #Lista_ComVel[11] := #Valor_B.low ;
           #Valor_W := #Valor_W * (-1);
           #Lista_ComVel[12] := #Valor_B.high ;
           #Lista_ComVel[13] := #Valor_B.low ;
           (* classic code: #Valor_W := REAL_TO_INT (#Valor_V3 * 163.84) ;*)
           #Valor_W := REAL_TO_INT (#Valor_V3 * REAL#163.84) ;
           #Lista_ComVel[14] := #Valor_B.high ;
           #Lista_ComVel[15] := #Valor_B.low ;
           #Valor_W := #Valor_W * (-1);
           #Lista_ComVel[16] := #Valor_B.high ;
           #Lista_ComVel[17] := #Valor_B.low ;
           (* classic code: #Valor_W := REAL_TO_INT (#Valor_V4 * 163.84) ;*)
           #Valor_W := REAL_TO_INT (#Valor_V4 * REAL#163.84) ;
           #Lista_ComVel[18] := #Valor_B.high ;
           #Lista_ComVel[19] := #Valor_B.low ;
           #Valor_W := #Valor_W * (-1);
           #Lista_ComVel[20] := #Valor_B.high ;
           #Lista_ComVel[21] := #Valor_B.low ;
           (* classic code: #Valor_W := REAL_TO_INT (#Valor_V5 * 163.84) ;*)
           #Valor_W := REAL_TO_INT (#Valor_V5 * REAL#163.84) ;
           #Lista_ComVel[22] := #Valor_B.high ;
           #Lista_ComVel[23] := #Valor_B.low ;
           #Valor_W := #Valor_W * (-1);
           #Lista_ComVel[24] := #Valor_B.high ;
           #Lista_ComVel[25] := #Valor_B.low ;
           (* classic code: #Valor_W := REAL_TO_INT (#Valor_V6 * 163.84) ;*)
           #Valor_W := REAL_TO_INT (#Valor_V6 * REAL#163.84) ;
           #Lista_ComVel[26] := #Valor_B.high ;
           #Lista_ComVel[27] := #Valor_B.low ;
           #Valor_W := #Valor_W * (-1);
           #Lista_ComVel[28] := #Valor_B.high ;
           #Lista_ComVel[29] := #Valor_B.low ;
           (* classic code: #Valor_W := REAL_TO_INT (#Valor_V7 * 163.84) ;*)
           #Valor_W := REAL_TO_INT (#Valor_V7 * REAL#163.84) ;
           #Lista_ComVel[30] := #Valor_B.high ;
           #Lista_ComVel[31] := #Valor_B.low ;
           #Valor_W := #Valor_W * (-1);
           #Lista_ComVel[32] := #Valor_B.high ;
           #Lista_ComVel[33] := #Valor_B.low ;

           //cabecera envio Rampa
           #Lista_ComRampa[1] := 16#7D ;
           #Lista_ComRampa[2] := INT_TO_BYTE (#Num_Line - 1) ;
           #Lista_ComRampa[3] := 16#0B ;
           #Lista_ComRampa[4] := INT_TO_BYTE (#Num_Slave);  //Num Esclavo ASI
           #Lista_ComRampa[5] := 16#0A ;
           #Lista_ComRampa[6] := 16#0E ;
           //Rampa (nos deben meter la rampa en milisegundos (tiempo para ir de 0 a 50Hz), solo miramos que no sea negativa)
           #Valor_W := ABS (#Valor_Rampa) ;
           #Lista_ComRampa[7] := #Valor_B.high ;
           #Lista_ComRampa[8] := #Valor_B.low ;

           IF #Solo_Rampa THEN
               #Ciclo_envio := 4 ;
           ELSE 
               #Ciclo_envio := 1 ;
           END_IF;

           #Con_Error := false ;

       END_IF;

       IF NOT #Escritura THEN
           #Ciclo_envio := 0 ;
       END_IF;

       CASE #Ciclo_envio OF
           1 :
               // ESCRITURA COMANDO DE VELOCIDADES
               (* classic code: %AB (#Dir_GW_ASI_Com):P := #Lista_ComVel[1];*)
               POKE(area:=16#02,dbNumber:=0,byteOffset:=#Dir_GW_ASI_Com,value:=#Lista_ComVel[1])  ;
               FOR #i := 2 TO 32 BY 1 DO    //copiamos todo
                   (* classic code: %AB (#Dir_GW_ASI_Com + #i):P := #Lista_ComVel[#i + 1];*)
                   POKE(area:=16#02,dbNumber:=0,byteOffset:=#Dir_GW_ASI_Com + #i,value:=#Lista_ComVel[#i + 1])  ;
               END_FOR;

               #Ciclo_envio := 2 ;

           2 :
               // ENVIO COMANDO DE VELOCIDADES
               (* classic code: #Lista_ComVel[2] := #Lista_ComVel[2] OR (%EB (#Dir_GW_ASI_Com + 1):P AND 16#80 ) XOR 16#80;*)
               #Lista_ComVel[2] := #Lista_ComVel[2] OR (PEEK_BYTE(area:=16#01,dbNumber:=0,byteOffset:=#Dir_GW_ASI_Com + 1) AND 16#80 ) XOR 16#80;  //Con el AND miro el bit de toogle en entradas, y lo invierto con el XOR, para despues añadirlo con el OR al comando ya calculado 
               (* classic code: %AB (#Dir_GW_ASI_Com + 1):P := #Lista_ComVel[2];*)
               POKE(area:=16#02,dbNumber:=0,byteOffset:=#Dir_GW_ASI_Com + 1,value:=#Lista_ComVel[2])  ;    //Me guardo el comando completo para saber luego que valor hemos enviado en Toogle

               #Ciclo_envio := 3 ;

           3 :
               // COMPROBAR RESPUESTA A COMANDO DE VELOCIDADES
               (* classic code: IF (%EB (#Dir_GW_ASI_Com + 1):P AND 16#80) = (#Lista_ComVel[2] AND 16#80) THEN*)
               IF (PEEK_BYTE(area:=16#01,dbNumber:=0,byteOffset:=#Dir_GW_ASI_Com + 1) AND 16#80) = (#Lista_ComVel[2] AND 16#80) THEN    //Miro si ha cambiado el Toogle
                   (* classic code: IF (%EB (#Dir_GW_ASI_Com):P = #Lista_ComVel[1]) AND (%EB (#Dir_GW_ASI_Com + 2):P = #Lista_ComVel[3]) THEN*)
                   IF (PEEK_BYTE(area:=16#01,dbNumber:=0,byteOffset:=#Dir_GW_ASI_Com) = #Lista_ComVel[1]) AND (PEEK_BYTE(area:=16#01,dbNumber:=0,byteOffset:=#Dir_GW_ASI_Com + 2) = #Lista_ComVel[3]) THEN   //Miro si el comando de vuelta es igual
                       IF #Solo_Velocidades THEN
                           #Ciclo_envio := 0 ;  //se ha ejecutado el envio correctamente y no hay que enviar rampa
                       ELSE
                           #Ciclo_envio := 4 ;  //se ha ejecutado el envio correctamente y pasamos a enviar rampa 
                       END_IF; 
                       #Con_Error := false ;
                   ELSE
                       #Ciclo_envio := 0 ;  //NO se ha ejecutado el envio correctamente
                       #Con_Error := true ;
                   END_IF;
               END_IF;

           4 :
               // ESCRITURA COMANDO DE RAMPA

               (* classic code: %AB (#Dir_GW_ASI_Com):P := #Lista_ComRampa[1];*)
               POKE(area:=16#02,dbNumber:=0,byteOffset:=#Dir_GW_ASI_Com,value:=#Lista_ComRampa[1])  ;
               FOR #i := 2 TO 7 BY 1 DO    //copiamos todo
                   (* classic code: %AB (#Dir_GW_ASI_Com + #i):P := #Lista_ComRampa[#i + 1];*)
                   POKE(area:=16#02,dbNumber:=0,byteOffset:=#Dir_GW_ASI_Com + #i,value:=#Lista_ComRampa[#i + 1])  ;
               END_FOR;

               #Ciclo_envio := 5 ;

           5 :
               // ENVIO COMANDO DE RAMPA
               (* classic code: #Lista_ComRampa[2] := #Lista_ComRampa[2] OR (%EB (#Dir_GW_ASI_Com + 1):P AND 16#80 ) XOR 16#80;*)
               #Lista_ComRampa[2] := #Lista_ComRampa[2] OR (PEEK_BYTE(area:=16#01,dbNumber:=0,byteOffset:=#Dir_GW_ASI_Com + 1) AND 16#80 ) XOR 16#80;  //Con el AND miro el bit de toogle en entradas, y lo invierto con el XOR, para despues añadirlo con el OR al comando ya calculado 
               (* classic code: %AB (#Dir_GW_ASI_Com + 1):P := #Lista_ComRampa[2];*)
               POKE(area:=16#02,dbNumber:=0,byteOffset:=#Dir_GW_ASI_Com + 1,value:=#Lista_ComRampa[2])  ;    //Me guardo el comando completo para saber luego que valor hemos enviado en Toogle

               #Ciclo_envio := 6 ;

           6 :
               // COMPROBAR RESPUESTA A COMANDO DE RAMPA
               (* classic code: IF (%EB (#Dir_GW_ASI_Com + 1):P AND 16#80) = (#Lista_ComRampa[2] AND 16#80) THEN*)
               IF (PEEK_BYTE(area:=16#01,dbNumber:=0,byteOffset:=#Dir_GW_ASI_Com + 1) AND 16#80) = (#Lista_ComRampa[2] AND 16#80) THEN    //Miro si ha cambiado el Toogle
                   (* classic code: IF (%EB (#Dir_GW_ASI_Com):P = #Lista_ComRampa[1]) AND (%EB (#Dir_GW_ASI_Com + 2):P = #Lista_ComRampa[3]) THEN*)
                   IF (PEEK_BYTE(area:=16#01,dbNumber:=0,byteOffset:=#Dir_GW_ASI_Com) = #Lista_ComRampa[1]) AND (PEEK_BYTE(area:=16#01,dbNumber:=0,byteOffset:=#Dir_GW_ASI_Com + 2) = #Lista_ComRampa[3]) THEN   //Miro si el comando de vuelta es igual
                       #Con_Error := false ;
                   ELSE 
                       #Con_Error := true ;  //NO se ha ejecutado el envio correctamente
                   END_IF;
               #Ciclo_envio := 0 ;
               END_IF;

       ELSE:
           // REPOSO, normalmente Ciclo_envio = 0, pero para cualquier otro caso no contemplado hacemos lo mismo
           #Ciclo_envio := 0 ;
           #Finalizado := #Escritura;
       END_CASE;

       IF NOT #Escritura THEN 
                   (* classic code: %AB (#Dir_GW_ASI_Com):P := 16#00 ;*)
                   POKE(area:=16#02,dbNumber:=0,byteOffset:=#Dir_GW_ASI_Com,value:=DINT_TO_BYTE(16#00))   ;
                   (* classic code: %AB (#Dir_GW_ASI_Com + 2):P := 16#00 ;*)
                   POKE(area:=16#02,dbNumber:=0,byteOffset:=#Dir_GW_ASI_Com + 2,value:=DINT_TO_BYTE(16#00))   ;
                   (* classic code: %AB (#Dir_GW_ASI_Com + 1):P := %EB (#Dir_GW_ASI_Com + 1):P ;*)
                   POKE(area:=16#02,dbNumber:=0,byteOffset:=#Dir_GW_ASI_Com + 1,value:=PEEK_BYTE(area:=16#01,dbNumber:=0,byteOffset:=#Dir_GW_ASI_Com + 1))   ;
       END_IF ;

    //   FOR i := 1 TO 255 BY 1 DO    //para rellenar el DB1000 todo como el Movimot[0]
    //       "Conf_Movimot".Movimot[i]:="Conf_Movimot".Movimot[0];
    //   END_FOR;

       #Escritura_OLD := #Escritura;
END_FUNCTION_BLOCK

FUNCTION "FC401_Conector_Mx_a_TL" : Void   // FC401, LAD
{ S7_Optimized_Access := 'FALSE' }
AUTHOR : TLigero
NAME : 20130323
VERSION : 3.0
// stored: AutoNumber false, SetENOAutomatically false
   VAR_INPUT
      Mesa : UInt;   // Numero de mesa de la funcion de ligero
      AVTF_MAnt_Mx : Bool;   // marca de la función de tracking
      MAnt_Avance : Bool;   // avance del transportador de tracking
      MAnt_DescargaAct : Bool;   // marca de la función de tracking
      PTF_Mx_MSig : Bool;   // marca de la función ligero
      NXT_Avance : Bool;   // avance del transportador ligero
      Rearme_V_Separacion : Bool;
      V_Separacion_T0_1s : UDInt;
   END_VAR
   VAR_OUTPUT
      NXT_AVTF_Conector : Bool;   // aviso para la función de ligero
      NXT_Descarga_Act_conector : Bool;   // descarga para la función de ligero
      PRV_PTF_conector : Bool;   // permiso para la función de tracking
      PRV_FTF_conector : Bool;   // fin para la función de tracking
   END_VAR
   VAR_TEMP
      Separacion_OK : Bool;
   END_VAR
BEGIN

REGION Network 1: contador de separación
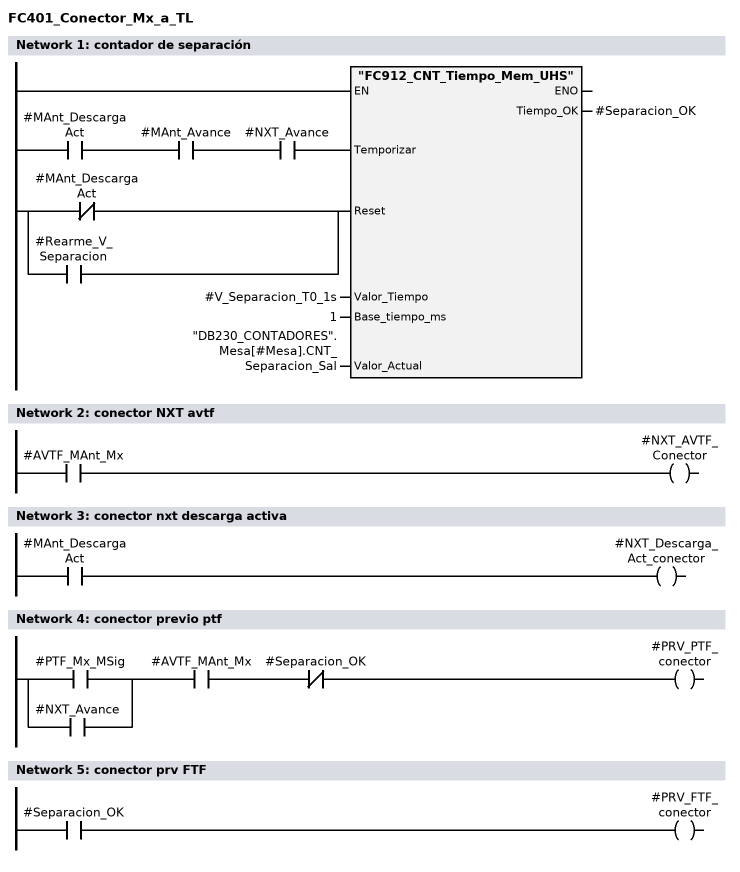
   RUNG wire#powerrail
      "FC912_CNT_Tiempo_Mem_UHS"(Temporizar := wire#w1, Reset := wire#w2, Valor_Tiempo := #V_Separacion_T0_1s, Base_tiempo_ms := 1, Valor_Actual := "DB230_CONTADORES".Mesa[#Mesa].CNT_Separacion_Sal, Tiempo_OK => #Separacion_OK)
   END_RUNG
   RUNG wire#powerrail
      Contact( #MAnt_DescargaAct )
      Contact( #MAnt_Avance )
      Contact( #NXT_Avance )
   END_RUNG wire#w1
   RUNG wire#powerrail
      I_Contact( #MAnt_DescargaAct )
   END_RUNG wire#w2
   RUNG wire#powerrail
      Contact( #Rearme_V_Separacion )
   END_RUNG wire#w2
   // the same network as SCL:
   "FC912_CNT_Tiempo_Mem_UHS"(Temporizar := #MAnt_DescargaAct AND #MAnt_Avance AND #NXT_Avance,
                           Reset := NOT #MAnt_DescargaAct OR #Rearme_V_Separacion,
                           Valor_Tiempo := #V_Separacion_T0_1s,
                           Base_tiempo_ms := 1,
                           Valor_Actual := "DB230_CONTADORES".Mesa[#Mesa].CNT_Separacion_Sal,
                           Tiempo_OK => #Separacion_OK);
END_REGION

REGION Network 2: conector NXT avtf
   RUNG wire#powerrail
      Contact( #AVTF_MAnt_Mx )
      Coil( #NXT_AVTF_Conector )
   END_RUNG
   // the same network as SCL:
   #NXT_AVTF_Conector := #AVTF_MAnt_Mx;
END_REGION

REGION Network 3: conector nxt descarga activa
   RUNG wire#powerrail
      Contact( #MAnt_DescargaAct )
      Coil( #NXT_Descarga_Act_conector )
   END_RUNG
   // the same network as SCL:
   #NXT_Descarga_Act_conector := #MAnt_DescargaAct;
END_REGION

REGION Network 4: conector previo ptf
   RUNG wire#powerrail
      Contact( #PTF_Mx_MSig )
      wire#w1
      Contact( #AVTF_MAnt_Mx )
      I_Contact( #Separacion_OK )
      Coil( #PRV_PTF_conector )
   END_RUNG
   RUNG wire#powerrail
      Contact( #NXT_Avance )
   END_RUNG wire#w1
   // the same network as SCL:
   #PRV_PTF_conector := (#PTF_Mx_MSig OR #NXT_Avance) AND #AVTF_MAnt_Mx AND NOT #Separacion_OK;
END_REGION

REGION Network 5: conector prv FTF
   RUNG wire#powerrail
      Contact( #Separacion_OK )
      Coil( #PRV_FTF_conector )
   END_RUNG
   // the same network as SCL:
   #PRV_FTF_conector := #Separacion_OK;
END_REGION
END_FUNCTION

FUNCTION "FC420_TL_ZPA_Tarjeta_CB" : Void   // FC420, LAD
{ S7_Optimized_Access := 'FALSE' }
AUTHOR : TLigero
NAME : 20160208
VERSION : 3.3
// stored: AutoNumber false, SetENOAutomatically false
   VAR_INPUT
      Mesa : UInt;
      En_Tension : Bool;
      PhsMx : Bool;
      Avance_Tx : Bool;
      Termico_Tx : Bool;
      Simul_Mx : Bool;
      AVTF_MAnt_Mx : Bool;
      PTF_Mx_MSig : Bool;
      NXT_Avance : Bool;
      V_Paro : UDInt;   // tiempo que avanza el transportador sin aviso hasta que se para (ms)
      V_TOut_Tx_Mx : UDInt;
      V_CNT_pHsMx : UDInt;
      V_Cara_Delantera : UDInt;   // valor separación entre caras delanteras (ms)
      V_Salida : UDInt;   // hueco mínimo entre cajas (ms)
      V_Gap : UDInt;   // espacio que se deja antes de iniciar un simultaneo
   END_VAR
   VAR_OUTPUT
      PTF_MAnt_Mx : Bool;
      AVTF_Mx_MSig : Bool;
      NXT_Descarga_Act : Bool;
   END_VAR
   VAR_IN_OUT
      Mem_CNT_Salida : Bool;
      Mem_CNT_Tmp_Paro_Tx : Bool;
      Maux_FP_Marcha : Bool;
      Maux_FN_PHS : Bool;
      MAux_Descarga_activa : Bool;
      Maux_permiso_paso : Bool;
      Maux_Tok : Bool;
      Maux_flanco : Bool;
   END_VAR
   VAR_TEMP
      OK_Avance : Bool;
      cara_delantera_OK : Bool;
      fp_Marcha : Bool;
      fn_phs_tx : Bool;
      fp_phs_tx : Bool;
      Mem_CNT_Centrado : Bool;
      Mem_CNT_Gap : Bool;
      Error_atasco : Bool;
      TEMP_NXT_AVTF : Bool;
      Reset_delantera : Bool;
      OK_tension : Bool;
   END_VAR
   VAR_TEMP   // added for the SCL form of the ladder/FBD networks
      _w1 : Bool;
   END_VAR
BEGIN

REGION Network 1: Marca General Error
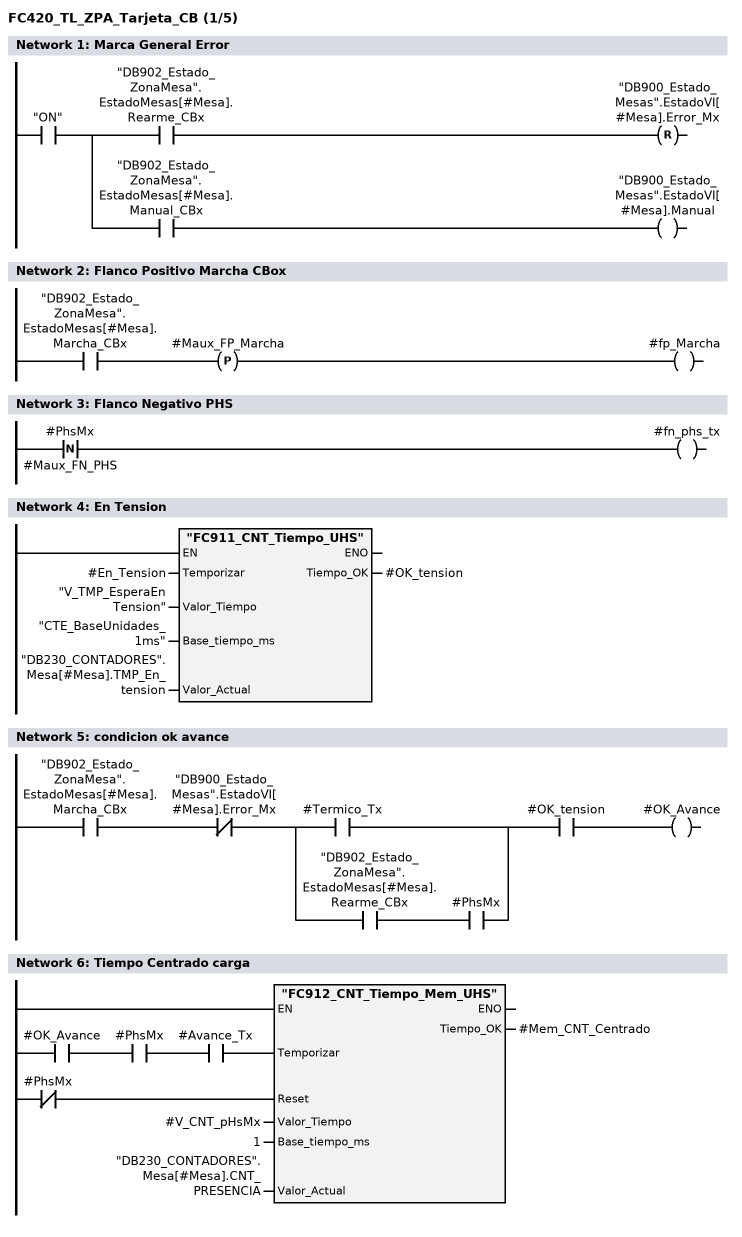
   RUNG wire#powerrail
      Contact( "ON" )
      wire#w1
      Contact( "DB902_Estado_ZonaMesa".EstadoMesas[#Mesa].Rearme_CBx )
      R_Coil( "DB900_Estado_Mesas".EstadoVI[#Mesa].Error_Mx )
   END_RUNG
   RUNG wire#w1
      Contact( "DB902_Estado_ZonaMesa".EstadoMesas[#Mesa].Manual_CBx )
      Coil( "DB900_Estado_Mesas".EstadoVI[#Mesa].Manual )
   END_RUNG
   // the same network as SCL:
   IF "ON" AND "DB902_Estado_ZonaMesa".EstadoMesas[#Mesa].Rearme_CBx THEN
       "DB900_Estado_Mesas".EstadoVI[#Mesa].Error_Mx := FALSE;
   END_IF;
   "DB900_Estado_Mesas".EstadoVI[#Mesa].Manual := "ON" AND "DB902_Estado_ZonaMesa".EstadoMesas[#Mesa].Manual_CBx;
END_REGION

REGION Network 2: Flanco Positivo Marcha CBox
   RUNG wire#powerrail
      Contact( "DB902_Estado_ZonaMesa".EstadoMesas[#Mesa].Marcha_CBx )
      P_Trig( #Maux_FP_Marcha )
      Coil( #fp_Marcha )
   END_RUNG
   // the same network as SCL:
   #_w1 := "DB902_Estado_ZonaMesa".EstadoMesas[#Mesa].Marcha_CBx AND NOT #Maux_FP_Marcha;   // rising edge
   #Maux_FP_Marcha := "DB902_Estado_ZonaMesa".EstadoMesas[#Mesa].Marcha_CBx;
   #fp_Marcha := #_w1;
END_REGION

REGION Network 3: Flanco Negativo PHS
   RUNG wire#powerrail
      N_Contact(operand := #PhsMx, bit := #Maux_FN_PHS)
      Coil( #fn_phs_tx )
   END_RUNG
   // the same network as SCL:
   #_w1 := NOT #PhsMx AND #Maux_FN_PHS;   // falling edge of #PhsMx
   #Maux_FN_PHS := #PhsMx;
   #fn_phs_tx := #_w1;
END_REGION

REGION Network 4: En Tension
   RUNG wire#powerrail
      "FC911_CNT_Tiempo_UHS"(Temporizar := #En_Tension, Valor_Tiempo := "V_TMP_EsperaEnTension", Base_tiempo_ms := "CTE_BaseUnidades_1ms", Valor_Actual := "DB230_CONTADORES".Mesa[#Mesa].TMP_En_tension, Tiempo_OK => #OK_tension)
   END_RUNG
   // the same network as SCL:
   "FC911_CNT_Tiempo_UHS"(Temporizar := #En_Tension,
                          Valor_Tiempo := "V_TMP_EsperaEnTension",
                          Base_tiempo_ms := "CTE_BaseUnidades_1ms",
                          Valor_Actual := "DB230_CONTADORES".Mesa[#Mesa].TMP_En_tension,
                          Tiempo_OK => #OK_tension);
END_REGION

REGION Network 5: condicion ok avance
   RUNG wire#powerrail
      Contact( "DB902_Estado_ZonaMesa".EstadoMesas[#Mesa].Marcha_CBx )
      I_Contact( "DB900_Estado_Mesas".EstadoVI[#Mesa].Error_Mx )
      wire#w1
      Contact( #Termico_Tx )
      wire#w2
      Contact( #OK_tension )
      Coil( #OK_Avance )
   END_RUNG
   RUNG wire#w1
      Contact( "DB902_Estado_ZonaMesa".EstadoMesas[#Mesa].Rearme_CBx )
      Contact( #PhsMx )
   END_RUNG wire#w2
   // the same network as SCL:
   #OK_Avance := "DB902_Estado_ZonaMesa".EstadoMesas[#Mesa].Marcha_CBx AND NOT "DB900_Estado_Mesas".EstadoVI[#Mesa].Error_Mx AND (#Termico_Tx OR ("DB902_Estado_ZonaMesa".EstadoMesas[#Mesa].Rearme_CBx AND #PhsMx)) AND #OK_tension;
END_REGION

REGION Network 6: Tiempo Centrado carga
   RUNG wire#powerrail
      "FC912_CNT_Tiempo_Mem_UHS"(Temporizar := wire#w1, Reset := wire#w2, Valor_Tiempo := #V_CNT_pHsMx, Base_tiempo_ms := 1, Valor_Actual := "DB230_CONTADORES".Mesa[#Mesa].CNT_PRESENCIA, Tiempo_OK => #Mem_CNT_Centrado)
   END_RUNG
   RUNG wire#powerrail
      Contact( #OK_Avance )
      Contact( #PhsMx )
      Contact( #Avance_Tx )
   END_RUNG wire#w1
   RUNG wire#powerrail
      I_Contact( #PhsMx )
   END_RUNG wire#w2
   // the same network as SCL:
   "FC912_CNT_Tiempo_Mem_UHS"(Temporizar := #OK_Avance AND #PhsMx AND #Avance_Tx,
                           Reset := NOT #PhsMx,
                           Valor_Tiempo := #V_CNT_pHsMx,
                           Base_tiempo_ms := 1,
                           Valor_Actual := "DB230_CONTADORES".Mesa[#Mesa].CNT_PRESENCIA,
                           Tiempo_OK => #Mem_CNT_Centrado);
END_REGION

REGION Network 7: contador tiempo de gap
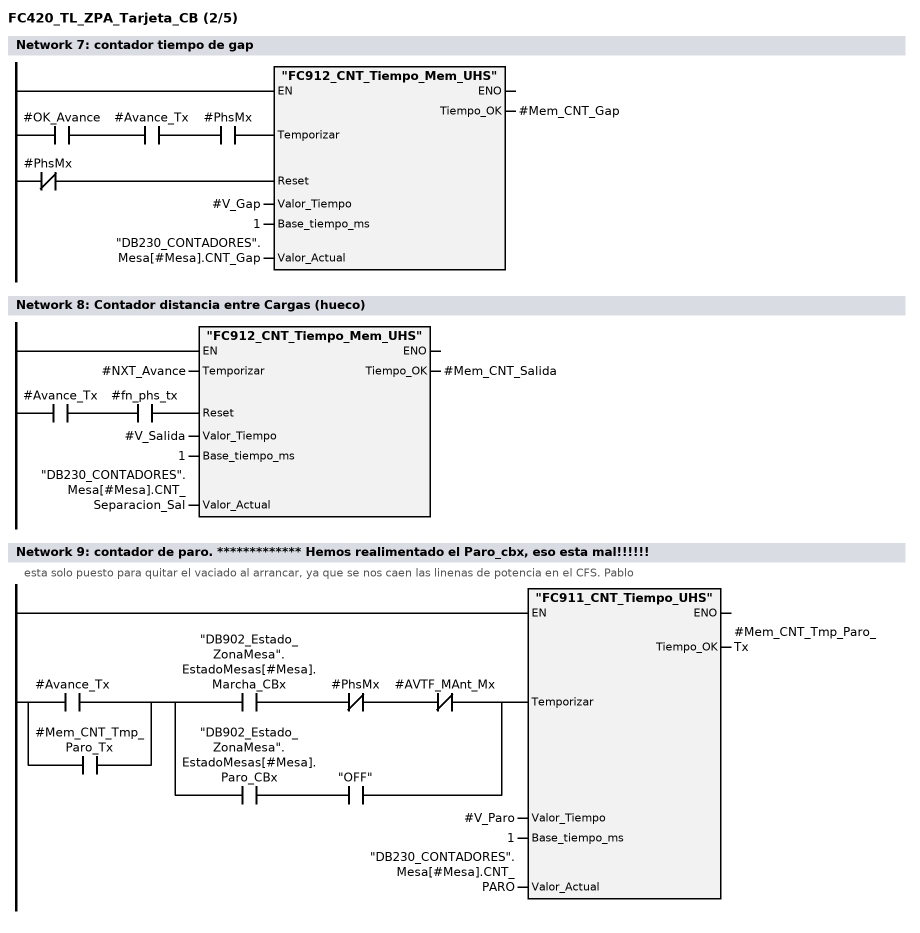
   RUNG wire#powerrail
      "FC912_CNT_Tiempo_Mem_UHS"(Temporizar := wire#w1, Reset := wire#w2, Valor_Tiempo := #V_Gap, Base_tiempo_ms := 1, Valor_Actual := "DB230_CONTADORES".Mesa[#Mesa].CNT_Gap, Tiempo_OK => #Mem_CNT_Gap)
   END_RUNG
   RUNG wire#powerrail
      Contact( #OK_Avance )
      Contact( #Avance_Tx )
      Contact( #PhsMx )
   END_RUNG wire#w1
   RUNG wire#powerrail
      I_Contact( #PhsMx )
   END_RUNG wire#w2
   // the same network as SCL:
   "FC912_CNT_Tiempo_Mem_UHS"(Temporizar := #OK_Avance AND #Avance_Tx AND #PhsMx,
                           Reset := NOT #PhsMx,
                           Valor_Tiempo := #V_Gap,
                           Base_tiempo_ms := 1,
                           Valor_Actual := "DB230_CONTADORES".Mesa[#Mesa].CNT_Gap,
                           Tiempo_OK => #Mem_CNT_Gap);
END_REGION

REGION Network 8: Contador distancia entre Cargas (hueco)
   RUNG wire#powerrail
      "FC912_CNT_Tiempo_Mem_UHS"(Reset := wire#w1, Temporizar := #NXT_Avance, Valor_Tiempo := #V_Salida, Base_tiempo_ms := 1, Valor_Actual := "DB230_CONTADORES".Mesa[#Mesa].CNT_Separacion_Sal, Tiempo_OK => #Mem_CNT_Salida)
   END_RUNG
   RUNG wire#powerrail
      Contact( #Avance_Tx )
      Contact( #fn_phs_tx )
   END_RUNG wire#w1
   // the same network as SCL:
   "FC912_CNT_Tiempo_Mem_UHS"(Temporizar := #NXT_Avance,
                           Reset := #Avance_Tx AND #fn_phs_tx,
                           Valor_Tiempo := #V_Salida,
                           Base_tiempo_ms := 1,
                           Valor_Actual := "DB230_CONTADORES".Mesa[#Mesa].CNT_Separacion_Sal,
                           Tiempo_OK => #Mem_CNT_Salida);
END_REGION

REGION Network 9: contador de paro. ************* Hemos realimentado el Paro_cbx, eso esta mal!!!!!!
   // esta solo puesto para quitar el vaciado al arrancar, ya que se nos caen las linenas de potencia en el CFS. Pablo
   RUNG wire#powerrail
      "FC911_CNT_Tiempo_UHS"(Temporizar := wire#w2, Valor_Tiempo := #V_Paro, Base_tiempo_ms := 1, Valor_Actual := "DB230_CONTADORES".Mesa[#Mesa].CNT_PARO, Tiempo_OK => #Mem_CNT_Tmp_Paro_Tx)
   END_RUNG
   RUNG wire#powerrail
      Contact( #Avance_Tx )
      wire#w1
      Contact( "DB902_Estado_ZonaMesa".EstadoMesas[#Mesa].Marcha_CBx )
      I_Contact( #PhsMx )
      I_Contact( #AVTF_MAnt_Mx )
   END_RUNG wire#w2
   RUNG wire#powerrail
      Contact( #Mem_CNT_Tmp_Paro_Tx )
   END_RUNG wire#w1
   RUNG wire#w1
      Contact( "DB902_Estado_ZonaMesa".EstadoMesas[#Mesa].Paro_CBx )
      Contact( "OFF" )
   END_RUNG wire#w2
   // the same network as SCL:
   "FC911_CNT_Tiempo_UHS"(Temporizar := (#Avance_Tx OR #Mem_CNT_Tmp_Paro_Tx) AND (("DB902_Estado_ZonaMesa".EstadoMesas[#Mesa].Marcha_CBx AND NOT #PhsMx AND NOT #AVTF_MAnt_Mx) OR ("DB902_Estado_ZonaMesa".EstadoMesas[#Mesa].Paro_CBx AND "OFF")),
                          Valor_Tiempo := #V_Paro,
                          Base_tiempo_ms := 1,
                          Valor_Actual := "DB230_CONTADORES".Mesa[#Mesa].CNT_PARO,
                          Tiempo_OK => #Mem_CNT_Tmp_Paro_Tx);
END_REGION

REGION Network 10: avance 13. QUITAMOS EL VACIADO PORQUE NOS SALTA LA FUENTE. SOLO EN CFS!!!!!!!!
   // ESTE SEGMENTO ESTA MAL!!! NNO DEBE ESTAR EL OFF EN EL FP_MARCHA. PABLO
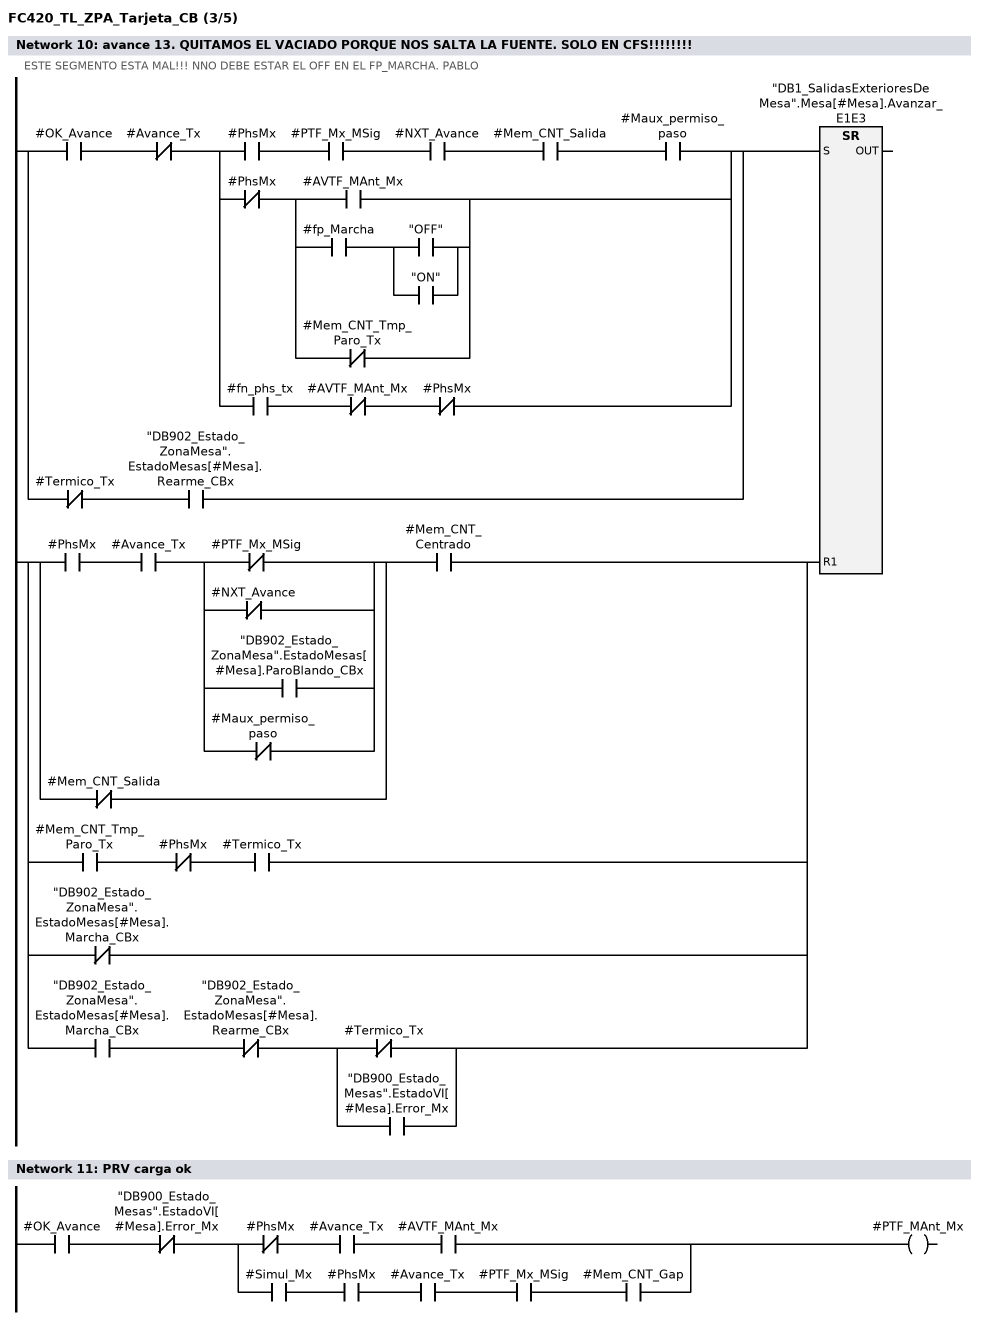
   RUNG wire#powerrail
      Contact( #OK_Avance )
      I_Contact( #Avance_Tx )
      wire#w1
      Contact( #PhsMx )
      Contact( #PTF_Mx_MSig )
      Contact( #NXT_Avance )
      Contact( #Mem_CNT_Salida )
      Contact( #Maux_permiso_paso )
      wire#w2
      S_SR(operand := "DB1_SalidasExterioresDeMesa".Mesa[#Mesa].Avanzar_E1E3, r1 := wire#w8)
   END_RUNG
   RUNG wire#w1
      I_Contact( #PhsMx )
      wire#w3
      Contact( #AVTF_MAnt_Mx )
   END_RUNG wire#w2
   RUNG wire#w3
      Contact( #fp_Marcha )
      wire#w4
      Contact( "OFF" )
   END_RUNG wire#w2
   RUNG wire#w4
      Contact( "ON" )
   END_RUNG wire#w2
   RUNG wire#w3
      I_Contact( #Mem_CNT_Tmp_Paro_Tx )
   END_RUNG wire#w2
   RUNG wire#w1
      Contact( #fn_phs_tx )
      I_Contact( #AVTF_MAnt_Mx )
      I_Contact( #PhsMx )
   END_RUNG wire#w2
   RUNG wire#powerrail
      I_Contact( #Termico_Tx )
      Contact( "DB902_Estado_ZonaMesa".EstadoMesas[#Mesa].Rearme_CBx )
   END_RUNG wire#w2
   RUNG wire#powerrail
      Contact( #PhsMx )
      Contact( #Avance_Tx )
      wire#w5
      I_Contact( #PTF_Mx_MSig )
      wire#w6
      Contact( #Mem_CNT_Centrado )
   END_RUNG wire#w8
   RUNG wire#w5
      I_Contact( #NXT_Avance )
   END_RUNG wire#w6
   RUNG wire#w5
      Contact( "DB902_Estado_ZonaMesa".EstadoMesas[#Mesa].ParoBlando_CBx )
   END_RUNG wire#w6
   RUNG wire#w5
      I_Contact( #Maux_permiso_paso )
   END_RUNG wire#w6
   RUNG wire#powerrail
      I_Contact( #Mem_CNT_Salida )
   END_RUNG wire#w6
   RUNG wire#powerrail
      Contact( #Mem_CNT_Tmp_Paro_Tx )
      I_Contact( #PhsMx )
      Contact( #Termico_Tx )
   END_RUNG wire#w8
   RUNG wire#powerrail
      I_Contact( "DB902_Estado_ZonaMesa".EstadoMesas[#Mesa].Marcha_CBx )
   END_RUNG wire#w8
   RUNG wire#powerrail
      Contact( "DB902_Estado_ZonaMesa".EstadoMesas[#Mesa].Marcha_CBx )
      I_Contact( "DB902_Estado_ZonaMesa".EstadoMesas[#Mesa].Rearme_CBx )
      wire#w7
      I_Contact( #Termico_Tx )
   END_RUNG wire#w8
   RUNG wire#w7
      Contact( "DB900_Estado_Mesas".EstadoVI[#Mesa].Error_Mx )
   END_RUNG wire#w8
   // the same network as SCL:
   #_w1 := (((#PhsMx AND #Avance_Tx AND (NOT #PTF_Mx_MSig OR NOT #NXT_Avance OR "DB902_Estado_ZonaMesa".EstadoMesas[#Mesa].ParoBlando_CBx OR NOT #Maux_permiso_paso)) OR NOT #Mem_CNT_Salida) AND #Mem_CNT_Centrado) OR (#Mem_CNT_Tmp_Paro_Tx AND NOT #PhsMx AND #Termico_Tx) OR NOT "DB902_Estado_ZonaMesa".EstadoMesas[#Mesa].Marcha_CBx OR ("DB902_Estado_ZonaMesa".EstadoMesas[#Mesa].Marcha_CBx AND NOT "DB902_Estado_ZonaMesa".EstadoMesas[#Mesa].Rearme_CBx AND (NOT #Termico_Tx OR "DB900_Estado_Mesas".EstadoVI[#Mesa].Error_Mx));
   IF (#OK_Avance AND NOT #Avance_Tx AND ((#PhsMx AND #PTF_Mx_MSig AND #NXT_Avance AND #Mem_CNT_Salida AND #Maux_permiso_paso) OR (NOT #PhsMx AND (#AVTF_MAnt_Mx OR (#fp_Marcha AND ("OFF" OR "ON")) OR NOT #Mem_CNT_Tmp_Paro_Tx)) OR (#fn_phs_tx AND NOT #AVTF_MAnt_Mx AND NOT #PhsMx))) OR (NOT #Termico_Tx AND "DB902_Estado_ZonaMesa".EstadoMesas[#Mesa].Rearme_CBx) THEN
       "DB1_SalidasExterioresDeMesa".Mesa[#Mesa].Avanzar_E1E3 := TRUE;   // SR flip-flop
   END_IF;
   IF #_w1 THEN "DB1_SalidasExterioresDeMesa".Mesa[#Mesa].Avanzar_E1E3 := FALSE; END_IF;
END_REGION

REGION Network 11: PRV carga ok
   RUNG wire#powerrail
      Contact( #OK_Avance )
      I_Contact( "DB900_Estado_Mesas".EstadoVI[#Mesa].Error_Mx )
      wire#w1
      I_Contact( #PhsMx )
      Contact( #Avance_Tx )
      Contact( #AVTF_MAnt_Mx )
      wire#w2
      Coil( #PTF_MAnt_Mx )
   END_RUNG
   RUNG wire#w1
      Contact( #Simul_Mx )
      Contact( #PhsMx )
      Contact( #Avance_Tx )
      Contact( #PTF_Mx_MSig )
      Contact( #Mem_CNT_Gap )
   END_RUNG wire#w2
   // the same network as SCL:
   #PTF_MAnt_Mx := #OK_Avance AND NOT "DB900_Estado_Mesas".EstadoVI[#Mesa].Error_Mx AND ((NOT #PhsMx AND #Avance_Tx AND #AVTF_MAnt_Mx) OR (#Simul_Mx AND #PhsMx AND #Avance_Tx AND #PTF_Mx_MSig AND #Mem_CNT_Gap));
END_REGION

REGION Network 12: NXT AVTF
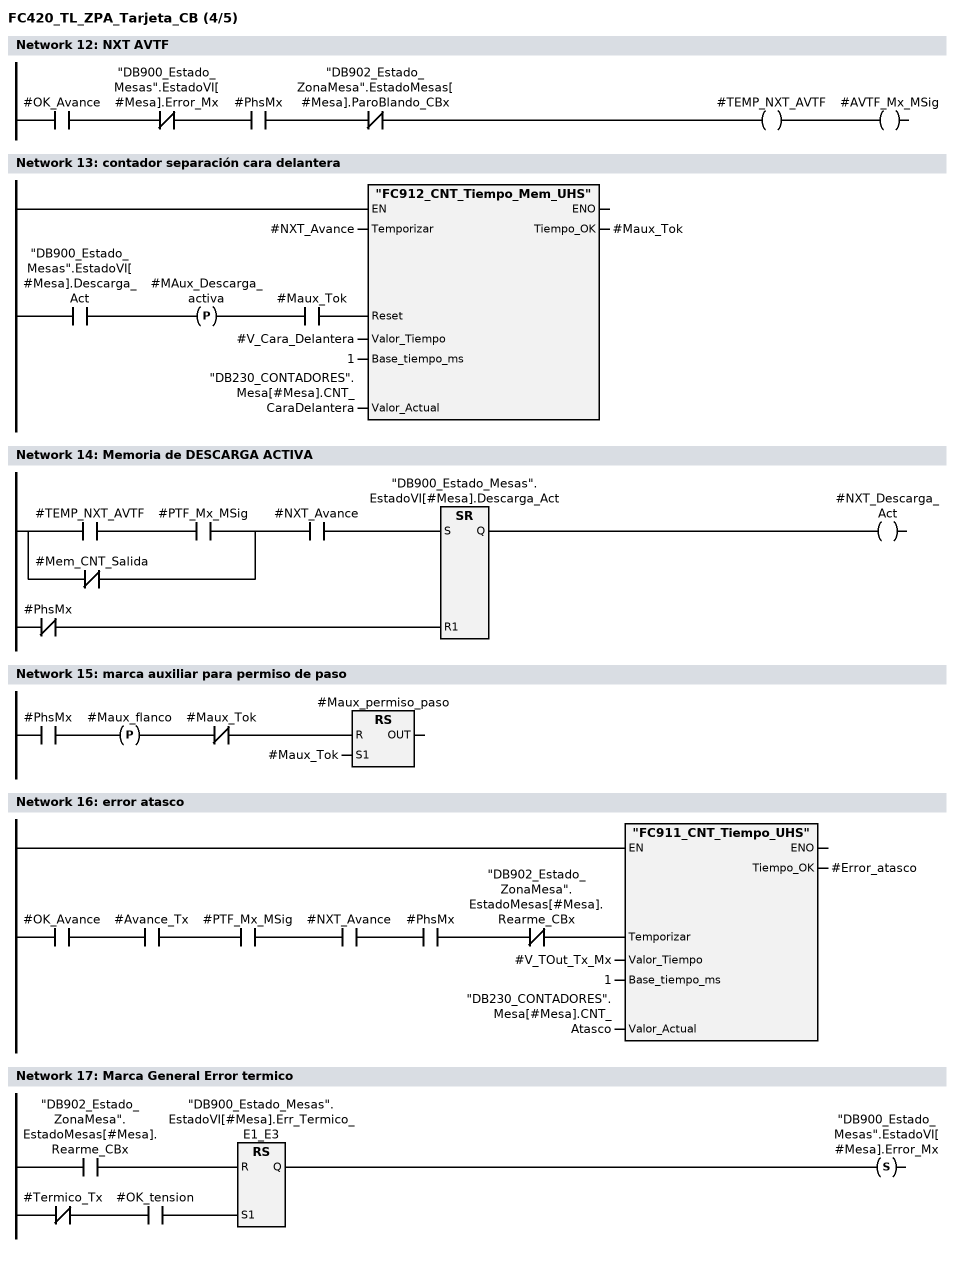
   RUNG wire#powerrail
      Contact( #OK_Avance )
      I_Contact( "DB900_Estado_Mesas".EstadoVI[#Mesa].Error_Mx )
      Contact( #PhsMx )
      I_Contact( "DB902_Estado_ZonaMesa".EstadoMesas[#Mesa].ParoBlando_CBx )
      Coil( #TEMP_NXT_AVTF )
      Coil( #AVTF_Mx_MSig )
   END_RUNG
   // the same network as SCL:
   #TEMP_NXT_AVTF := #OK_Avance AND NOT "DB900_Estado_Mesas".EstadoVI[#Mesa].Error_Mx AND #PhsMx AND NOT "DB902_Estado_ZonaMesa".EstadoMesas[#Mesa].ParoBlando_CBx;
   #AVTF_Mx_MSig := #TEMP_NXT_AVTF;
END_REGION

REGION Network 13: contador separación cara delantera
   RUNG wire#powerrail
      "FC912_CNT_Tiempo_Mem_UHS"(Reset := wire#w1, Temporizar := #NXT_Avance, Valor_Tiempo := #V_Cara_Delantera, Base_tiempo_ms := 1, Valor_Actual := "DB230_CONTADORES".Mesa[#Mesa].CNT_CaraDelantera, Tiempo_OK => #Maux_Tok)
   END_RUNG
   RUNG wire#powerrail
      Contact( "DB900_Estado_Mesas".EstadoVI[#Mesa].Descarga_Act )
      P_Trig( #MAux_Descarga_activa )
      Contact( #Maux_Tok )
   END_RUNG wire#w1
   // the same network as SCL:
   #_w1 := "DB900_Estado_Mesas".EstadoVI[#Mesa].Descarga_Act AND NOT #MAux_Descarga_activa;   // rising edge
   #MAux_Descarga_activa := "DB900_Estado_Mesas".EstadoVI[#Mesa].Descarga_Act;
   "FC912_CNT_Tiempo_Mem_UHS"(Temporizar := #NXT_Avance,
                           Reset := #_w1 AND #Maux_Tok,
                           Valor_Tiempo := #V_Cara_Delantera,
                           Base_tiempo_ms := 1,
                           Valor_Actual := "DB230_CONTADORES".Mesa[#Mesa].CNT_CaraDelantera,
                           Tiempo_OK => #Maux_Tok);
END_REGION

REGION Network 14: Memoria de DESCARGA ACTIVA
   RUNG wire#powerrail
      Contact( #TEMP_NXT_AVTF )
      Contact( #PTF_Mx_MSig )
      wire#w1
      Contact( #NXT_Avance )
      S_SR(operand := "DB900_Estado_Mesas".EstadoVI[#Mesa].Descarga_Act, r1 := wire#w2)
      Coil( #NXT_Descarga_Act )
   END_RUNG
   RUNG wire#powerrail
      I_Contact( #Mem_CNT_Salida )
   END_RUNG wire#w1
   RUNG wire#powerrail
      I_Contact( #PhsMx )
   END_RUNG wire#w2
   // the same network as SCL:
   IF ((#TEMP_NXT_AVTF AND #PTF_Mx_MSig) OR NOT #Mem_CNT_Salida) AND #NXT_Avance THEN
       "DB900_Estado_Mesas".EstadoVI[#Mesa].Descarga_Act := TRUE;   // SR flip-flop
   END_IF;
   IF NOT #PhsMx THEN "DB900_Estado_Mesas".EstadoVI[#Mesa].Descarga_Act := FALSE; END_IF;
   #NXT_Descarga_Act := "DB900_Estado_Mesas".EstadoVI[#Mesa].Descarga_Act;
END_REGION

REGION Network 15: marca auxiliar para permiso de paso
   RUNG wire#powerrail
      Contact( #PhsMx )
      P_Trig( #Maux_flanco )
      I_Contact( #Maux_Tok )
      S_RS(operand := #Maux_permiso_paso, s1 := #Maux_Tok)
   END_RUNG
   // the same network as SCL:
   #_w1 := #PhsMx AND NOT #Maux_flanco;   // rising edge
   #Maux_flanco := #PhsMx;
   IF #_w1 AND NOT #Maux_Tok THEN
       #Maux_permiso_paso := FALSE;   // RS flip-flop
   END_IF;
   IF #Maux_Tok THEN #Maux_permiso_paso := TRUE; END_IF;
END_REGION

REGION Network 16: error atasco
   RUNG wire#powerrail
      "FC911_CNT_Tiempo_UHS"(Temporizar := wire#w1, Valor_Tiempo := #V_TOut_Tx_Mx, Base_tiempo_ms := 1, Valor_Actual := "DB230_CONTADORES".Mesa[#Mesa].CNT_Atasco, Tiempo_OK => #Error_atasco)
   END_RUNG
   RUNG wire#powerrail
      Contact( #OK_Avance )
      Contact( #Avance_Tx )
      Contact( #PTF_Mx_MSig )
      Contact( #NXT_Avance )
      Contact( #PhsMx )
      I_Contact( "DB902_Estado_ZonaMesa".EstadoMesas[#Mesa].Rearme_CBx )
   END_RUNG wire#w1
   // the same network as SCL:
   "FC911_CNT_Tiempo_UHS"(Temporizar := #OK_Avance AND #Avance_Tx AND #PTF_Mx_MSig AND #NXT_Avance AND #PhsMx AND NOT "DB902_Estado_ZonaMesa".EstadoMesas[#Mesa].Rearme_CBx,
                          Valor_Tiempo := #V_TOut_Tx_Mx,
                          Base_tiempo_ms := 1,
                          Valor_Actual := "DB230_CONTADORES".Mesa[#Mesa].CNT_Atasco,
                          Tiempo_OK => #Error_atasco);
END_REGION

REGION Network 17: Marca General Error termico
   RUNG wire#powerrail
      Contact( "DB902_Estado_ZonaMesa".EstadoMesas[#Mesa].Rearme_CBx )
      S_RS(operand := "DB900_Estado_Mesas".EstadoVI[#Mesa].Err_Termico_E1_E3, s1 := wire#w1)
      S_Coil( "DB900_Estado_Mesas".EstadoVI[#Mesa].Error_Mx )
   END_RUNG
   RUNG wire#powerrail
      I_Contact( #Termico_Tx )
      Contact( #OK_tension )
   END_RUNG wire#w1
   // the same network as SCL:
   IF "DB902_Estado_ZonaMesa".EstadoMesas[#Mesa].Rearme_CBx THEN
       "DB900_Estado_Mesas".EstadoVI[#Mesa].Err_Termico_E1_E3 := FALSE;   // RS flip-flop
   END_IF;
   IF NOT #Termico_Tx AND #OK_tension THEN
       "DB900_Estado_Mesas".EstadoVI[#Mesa].Err_Termico_E1_E3 := TRUE;
   END_IF;
   IF "DB900_Estado_Mesas".EstadoVI[#Mesa].Err_Termico_E1_E3 THEN
       "DB900_Estado_Mesas".EstadoVI[#Mesa].Error_Mx := TRUE;
   END_IF;
END_REGION

REGION Network 18: Marca General Error tout avance
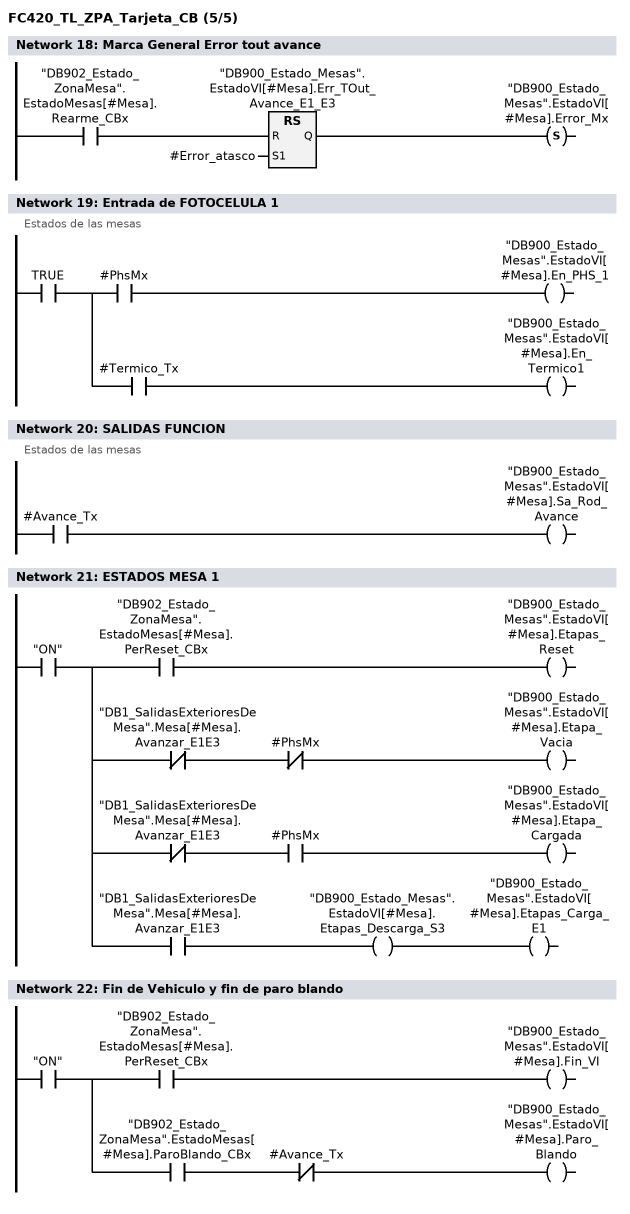
   RUNG wire#powerrail
      Contact( "DB902_Estado_ZonaMesa".EstadoMesas[#Mesa].Rearme_CBx )
      S_RS(operand := "DB900_Estado_Mesas".EstadoVI[#Mesa].Err_TOut_Avance_E1_E3, s1 := #Error_atasco)
      S_Coil( "DB900_Estado_Mesas".EstadoVI[#Mesa].Error_Mx )
   END_RUNG
   // the same network as SCL:
   IF "DB902_Estado_ZonaMesa".EstadoMesas[#Mesa].Rearme_CBx THEN
       "DB900_Estado_Mesas".EstadoVI[#Mesa].Err_TOut_Avance_E1_E3 := FALSE;   // RS flip-flop
   END_IF;
   IF #Error_atasco THEN "DB900_Estado_Mesas".EstadoVI[#Mesa].Err_TOut_Avance_E1_E3 := TRUE; END_IF;
   IF "DB900_Estado_Mesas".EstadoVI[#Mesa].Err_TOut_Avance_E1_E3 THEN
       "DB900_Estado_Mesas".EstadoVI[#Mesa].Error_Mx := TRUE;
   END_IF;
END_REGION

REGION Network 19: Entrada de FOTOCELULA 1
   // Estados de las mesas
   RUNG wire#powerrail
      Contact( TRUE )
      wire#w1
      Contact( #PhsMx )
      Coil( "DB900_Estado_Mesas".EstadoVI[#Mesa].En_PHS_1 )
   END_RUNG
   RUNG wire#w1
      Contact( #Termico_Tx )
      Coil( "DB900_Estado_Mesas".EstadoVI[#Mesa].En_Termico1 )
   END_RUNG
   // the same network as SCL:
   "DB900_Estado_Mesas".EstadoVI[#Mesa].En_PHS_1 := TRUE AND #PhsMx;
   "DB900_Estado_Mesas".EstadoVI[#Mesa].En_Termico1 := TRUE AND #Termico_Tx;
END_REGION

REGION Network 20: SALIDAS FUNCION
   // Estados de las mesas
   RUNG wire#powerrail
      Contact( #Avance_Tx )
      Coil( "DB900_Estado_Mesas".EstadoVI[#Mesa].Sa_Rod_Avance )
   END_RUNG
   // the same network as SCL:
   "DB900_Estado_Mesas".EstadoVI[#Mesa].Sa_Rod_Avance := #Avance_Tx;
END_REGION

REGION Network 21: ESTADOS MESA 1
   RUNG wire#powerrail
      Contact( "ON" )
      wire#w1
      Contact( "DB902_Estado_ZonaMesa".EstadoMesas[#Mesa].PerReset_CBx )
      Coil( "DB900_Estado_Mesas".EstadoVI[#Mesa].Etapas_Reset )
   END_RUNG
   RUNG wire#w1
      I_Contact( "DB1_SalidasExterioresDeMesa".Mesa[#Mesa].Avanzar_E1E3 )
      I_Contact( #PhsMx )
      Coil( "DB900_Estado_Mesas".EstadoVI[#Mesa].Etapa_Vacia )
   END_RUNG
   RUNG wire#w1
      I_Contact( "DB1_SalidasExterioresDeMesa".Mesa[#Mesa].Avanzar_E1E3 )
      Contact( #PhsMx )
      Coil( "DB900_Estado_Mesas".EstadoVI[#Mesa].Etapa_Cargada )
   END_RUNG
   RUNG wire#w1
      Contact( "DB1_SalidasExterioresDeMesa".Mesa[#Mesa].Avanzar_E1E3 )
      Coil( "DB900_Estado_Mesas".EstadoVI[#Mesa].Etapas_Descarga_S3 )
      Coil( "DB900_Estado_Mesas".EstadoVI[#Mesa].Etapas_Carga_E1 )
   END_RUNG
   // the same network as SCL:
   "DB900_Estado_Mesas".EstadoVI[#Mesa].Etapas_Reset := "ON" AND "DB902_Estado_ZonaMesa".EstadoMesas[#Mesa].PerReset_CBx;
   "DB900_Estado_Mesas".EstadoVI[#Mesa].Etapa_Vacia := "ON" AND NOT "DB1_SalidasExterioresDeMesa".Mesa[#Mesa].Avanzar_E1E3 AND NOT #PhsMx;
   "DB900_Estado_Mesas".EstadoVI[#Mesa].Etapa_Cargada := "ON" AND NOT "DB1_SalidasExterioresDeMesa".Mesa[#Mesa].Avanzar_E1E3 AND #PhsMx;
   #_w1 := "ON" AND "DB1_SalidasExterioresDeMesa".Mesa[#Mesa].Avanzar_E1E3;
   "DB900_Estado_Mesas".EstadoVI[#Mesa].Etapas_Descarga_S3 := #_w1;
   "DB900_Estado_Mesas".EstadoVI[#Mesa].Etapas_Carga_E1 := #_w1;
END_REGION

REGION Network 22: Fin de Vehiculo y fin de paro blando
   RUNG wire#powerrail
      Contact( "ON" )
      wire#w1
      Contact( "DB902_Estado_ZonaMesa".EstadoMesas[#Mesa].PerReset_CBx )
      Coil( "DB900_Estado_Mesas".EstadoVI[#Mesa].Fin_VI )
   END_RUNG
   RUNG wire#w1
      Contact( "DB902_Estado_ZonaMesa".EstadoMesas[#Mesa].ParoBlando_CBx )
      I_Contact( #Avance_Tx )
      Coil( "DB900_Estado_Mesas".EstadoVI[#Mesa].Paro_Blando )
   END_RUNG
   // the same network as SCL:
   "DB900_Estado_Mesas".EstadoVI[#Mesa].Fin_VI := "ON" AND "DB902_Estado_ZonaMesa".EstadoMesas[#Mesa].PerReset_CBx;
   "DB900_Estado_Mesas".EstadoVI[#Mesa].Paro_Blando := "ON" AND "DB902_Estado_ZonaMesa".EstadoMesas[#Mesa].ParoBlando_CBx AND NOT #Avance_Tx;
END_REGION
END_FUNCTION

FUNCTION "FC450_TL_TR_E1_S2_Pres" : Void   // FC450, LAD
{ S7_Optimized_Access := 'FALSE' }
AUTHOR : TLigero
NAME : 20160512
VERSION : 4.0
// stored: AutoNumber false, SetENOAutomatically false
   VAR_INPUT
      Mesa : UInt;
      En_Tension : Bool;
      PhsMx : Bool;
      Termico_E1 : Bool;
      Termico_S2 : Bool;
      PosTR_E1 : Bool;
      PosTR_S2 : Bool;
      Avance_E1 : Bool;
      Avance_S2 : Bool;
      AVTF_MAnt_Mx : Bool;   // Aviso de transferencia de la mesa anterior
      PTF_Mx_MSig : Bool;   // Permiso de transferencia de la mesa siguiente
      NXT_Avance : Bool;   // Avance de la mesa siguiente
      V_CNT_pHsMx : UDInt;
      V_CNT_ApHsMx : UDInt;
      V_Paro : UDInt;
      V_TOut_Tx_Mx : UDInt;
      V_TOut_transfer : UDInt;
   END_VAR
   VAR_OUTPUT
      PTF_MAnt_Mx : Bool;   // carga ok a la mesa anterior
      AVTF_Mx_MSig : Bool;   // Aviso de transferencia a la mesa siguiente
      NXT_Descarga_Act : Bool;   // descarga activa a la mesa siguiente
   END_VAR
   VAR_TEMP
      Mem_CNT_Tmp_Paro_Tx : Bool;
      Mem_CNT_Pres_entrada : Bool;
      Mem_CNT_Aus_salida : Bool;
      tout_atasco : Bool;
      tout_transfer : Bool;
      TEMP_MA_TR_Pos_E1 : Bool;
      TEMP_MA_TR_Pos_S2 : Bool;
      ok_tension : Bool;
   END_VAR
   VAR_TEMP   // added for the SCL form of the ladder/FBD networks
      _w1 : Bool;
   END_VAR
BEGIN

REGION Network 1: Marca General Error
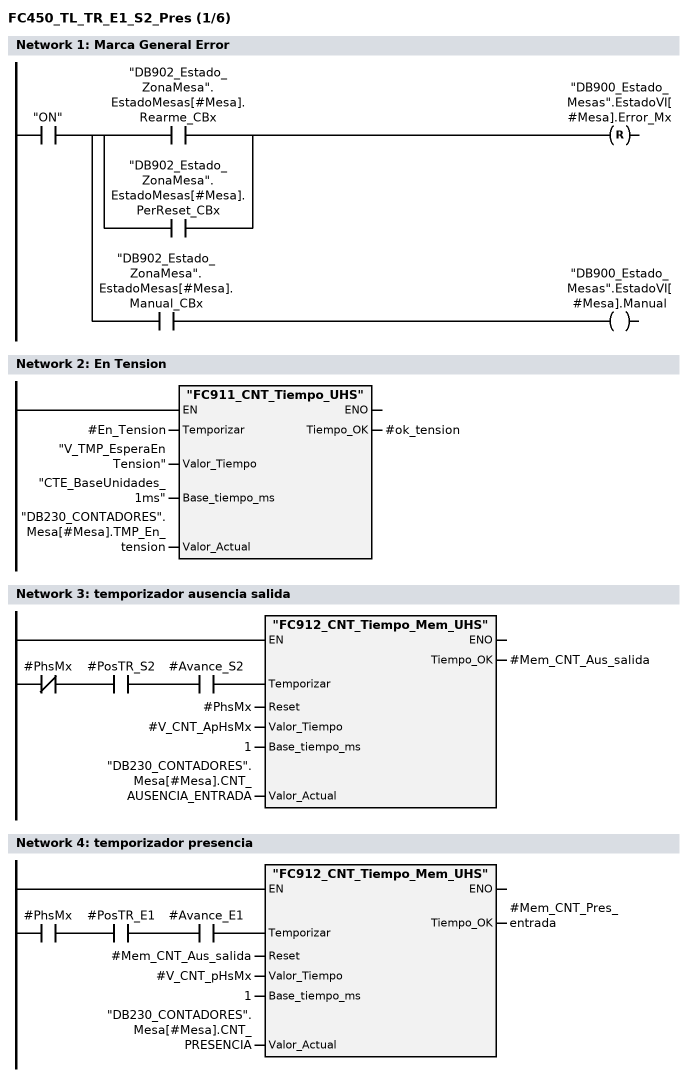
   RUNG wire#powerrail
      Contact( "ON" )
      wire#w1
      Contact( "DB902_Estado_ZonaMesa".EstadoMesas[#Mesa].Rearme_CBx )
      wire#w2
      R_Coil( "DB900_Estado_Mesas".EstadoVI[#Mesa].Error_Mx )
   END_RUNG
   RUNG wire#w1
      Contact( "DB902_Estado_ZonaMesa".EstadoMesas[#Mesa].PerReset_CBx )
   END_RUNG wire#w2
   RUNG wire#w1
      Contact( "DB902_Estado_ZonaMesa".EstadoMesas[#Mesa].Manual_CBx )
      Coil( "DB900_Estado_Mesas".EstadoVI[#Mesa].Manual )
   END_RUNG
   // the same network as SCL:
   IF "ON" AND ("DB902_Estado_ZonaMesa".EstadoMesas[#Mesa].Rearme_CBx OR "DB902_Estado_ZonaMesa".EstadoMesas[#Mesa].PerReset_CBx) THEN
       "DB900_Estado_Mesas".EstadoVI[#Mesa].Error_Mx := FALSE;
   END_IF;
   "DB900_Estado_Mesas".EstadoVI[#Mesa].Manual := "ON" AND "DB902_Estado_ZonaMesa".EstadoMesas[#Mesa].Manual_CBx;
END_REGION

REGION Network 2: En Tension
   RUNG wire#powerrail
      "FC911_CNT_Tiempo_UHS"(Temporizar := #En_Tension, Valor_Tiempo := "V_TMP_EsperaEnTension", Base_tiempo_ms := "CTE_BaseUnidades_1ms", Valor_Actual := "DB230_CONTADORES".Mesa[#Mesa].TMP_En_tension, Tiempo_OK => #ok_tension)
   END_RUNG
   // the same network as SCL:
   "FC911_CNT_Tiempo_UHS"(Temporizar := #En_Tension,
                          Valor_Tiempo := "V_TMP_EsperaEnTension",
                          Base_tiempo_ms := "CTE_BaseUnidades_1ms",
                          Valor_Actual := "DB230_CONTADORES".Mesa[#Mesa].TMP_En_tension,
                          Tiempo_OK => #ok_tension);
END_REGION

REGION Network 3: temporizador ausencia salida
   RUNG wire#powerrail
      "FC912_CNT_Tiempo_Mem_UHS"(Temporizar := wire#w1, Reset := #PhsMx, Valor_Tiempo := #V_CNT_ApHsMx, Base_tiempo_ms := 1, Valor_Actual := "DB230_CONTADORES".Mesa[#Mesa].CNT_AUSENCIA_ENTRADA, Tiempo_OK => #Mem_CNT_Aus_salida)
   END_RUNG
   RUNG wire#powerrail
      I_Contact( #PhsMx )
      Contact( #PosTR_S2 )
      Contact( #Avance_S2 )
   END_RUNG wire#w1
   // the same network as SCL:
   "FC912_CNT_Tiempo_Mem_UHS"(Temporizar := NOT #PhsMx AND #PosTR_S2 AND #Avance_S2,
                           Reset := #PhsMx,
                           Valor_Tiempo := #V_CNT_ApHsMx,
                           Base_tiempo_ms := 1,
                           Valor_Actual := "DB230_CONTADORES".Mesa[#Mesa].CNT_AUSENCIA_ENTRADA,
                           Tiempo_OK => #Mem_CNT_Aus_salida);
END_REGION

REGION Network 4: temporizador presencia
   RUNG wire#powerrail
      "FC912_CNT_Tiempo_Mem_UHS"(Temporizar := wire#w1, Reset := #Mem_CNT_Aus_salida, Valor_Tiempo := #V_CNT_pHsMx, Base_tiempo_ms := 1, Valor_Actual := "DB230_CONTADORES".Mesa[#Mesa].CNT_PRESENCIA, Tiempo_OK => #Mem_CNT_Pres_entrada)
   END_RUNG
   RUNG wire#powerrail
      Contact( #PhsMx )
      Contact( #PosTR_E1 )
      Contact( #Avance_E1 )
   END_RUNG wire#w1
   // the same network as SCL:
   "FC912_CNT_Tiempo_Mem_UHS"(Temporizar := #PhsMx AND #PosTR_E1 AND #Avance_E1,
                           Reset := #Mem_CNT_Aus_salida,
                           Valor_Tiempo := #V_CNT_pHsMx,
                           Base_tiempo_ms := 1,
                           Valor_Actual := "DB230_CONTADORES".Mesa[#Mesa].CNT_PRESENCIA,
                           Tiempo_OK => #Mem_CNT_Pres_entrada);
END_REGION

REGION Network 5: temporizador PARO
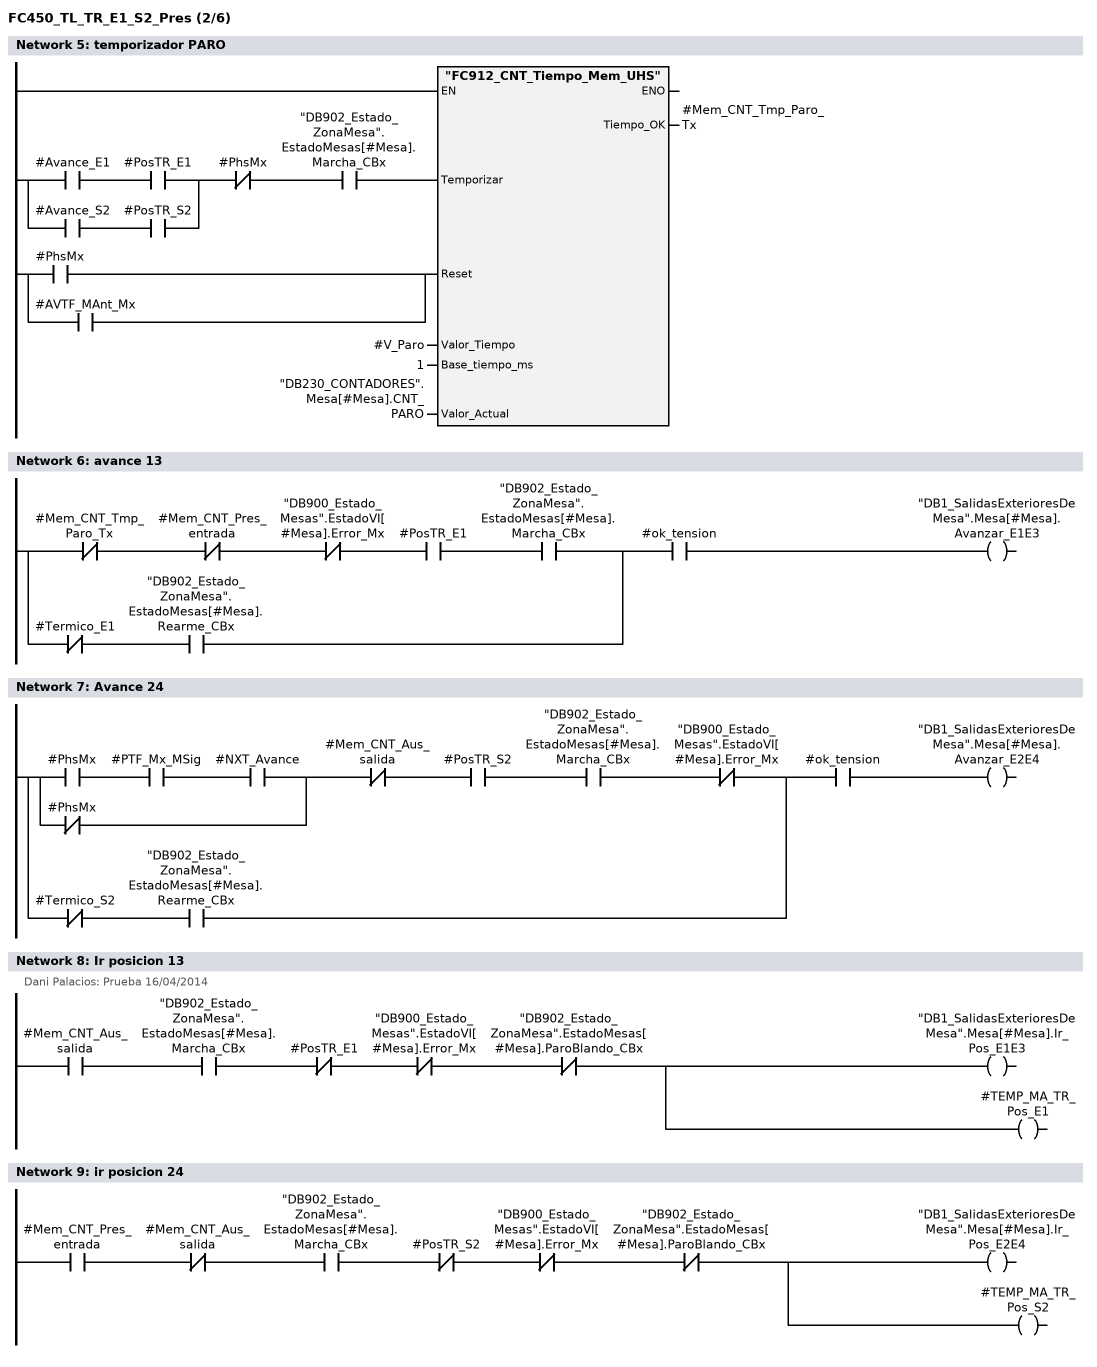
   RUNG wire#powerrail
      "FC912_CNT_Tiempo_Mem_UHS"(Temporizar := wire#w2, Reset := wire#w3, Valor_Tiempo := #V_Paro, Base_tiempo_ms := 1, Valor_Actual := "DB230_CONTADORES".Mesa[#Mesa].CNT_PARO, Tiempo_OK => #Mem_CNT_Tmp_Paro_Tx)
   END_RUNG
   RUNG wire#powerrail
      Contact( #Avance_E1 )
      Contact( #PosTR_E1 )
      wire#w1
      I_Contact( #PhsMx )
      Contact( "DB902_Estado_ZonaMesa".EstadoMesas[#Mesa].Marcha_CBx )
   END_RUNG wire#w2
   RUNG wire#powerrail
      Contact( #Avance_S2 )
      Contact( #PosTR_S2 )
   END_RUNG wire#w1
   RUNG wire#powerrail
      Contact( #PhsMx )
   END_RUNG wire#w3
   RUNG wire#powerrail
      Contact( #AVTF_MAnt_Mx )
   END_RUNG wire#w3
   // the same network as SCL:
   "FC912_CNT_Tiempo_Mem_UHS"(Temporizar := ((#Avance_E1 AND #PosTR_E1) OR (#Avance_S2 AND #PosTR_S2)) AND NOT #PhsMx AND "DB902_Estado_ZonaMesa".EstadoMesas[#Mesa].Marcha_CBx,
                           Reset := #PhsMx OR #AVTF_MAnt_Mx,
                           Valor_Tiempo := #V_Paro,
                           Base_tiempo_ms := 1,
                           Valor_Actual := "DB230_CONTADORES".Mesa[#Mesa].CNT_PARO,
                           Tiempo_OK => #Mem_CNT_Tmp_Paro_Tx);
END_REGION

REGION Network 6: avance 13
   RUNG wire#powerrail
      I_Contact( #Mem_CNT_Tmp_Paro_Tx )
      I_Contact( #Mem_CNT_Pres_entrada )
      I_Contact( "DB900_Estado_Mesas".EstadoVI[#Mesa].Error_Mx )
      Contact( #PosTR_E1 )
      Contact( "DB902_Estado_ZonaMesa".EstadoMesas[#Mesa].Marcha_CBx )
      wire#w1
      Contact( #ok_tension )
      Coil( "DB1_SalidasExterioresDeMesa".Mesa[#Mesa].Avanzar_E1E3 )
   END_RUNG
   RUNG wire#powerrail
      I_Contact( #Termico_E1 )
      Contact( "DB902_Estado_ZonaMesa".EstadoMesas[#Mesa].Rearme_CBx )
   END_RUNG wire#w1
   // the same network as SCL:
   "DB1_SalidasExterioresDeMesa".Mesa[#Mesa].Avanzar_E1E3 := ((NOT #Mem_CNT_Tmp_Paro_Tx AND NOT #Mem_CNT_Pres_entrada AND NOT "DB900_Estado_Mesas".EstadoVI[#Mesa].Error_Mx AND #PosTR_E1 AND "DB902_Estado_ZonaMesa".EstadoMesas[#Mesa].Marcha_CBx) OR (NOT #Termico_E1 AND "DB902_Estado_ZonaMesa".EstadoMesas[#Mesa].Rearme_CBx)) AND #ok_tension;
END_REGION

REGION Network 7: Avance 24
   RUNG wire#powerrail
      Contact( #PhsMx )
      Contact( #PTF_Mx_MSig )
      Contact( #NXT_Avance )
      wire#w1
      I_Contact( #Mem_CNT_Aus_salida )
      Contact( #PosTR_S2 )
      Contact( "DB902_Estado_ZonaMesa".EstadoMesas[#Mesa].Marcha_CBx )
      I_Contact( "DB900_Estado_Mesas".EstadoVI[#Mesa].Error_Mx )
      wire#w2
      Contact( #ok_tension )
      Coil( "DB1_SalidasExterioresDeMesa".Mesa[#Mesa].Avanzar_E2E4 )
   END_RUNG
   RUNG wire#powerrail
      I_Contact( #PhsMx )
   END_RUNG wire#w1
   RUNG wire#powerrail
      I_Contact( #Termico_S2 )
      Contact( "DB902_Estado_ZonaMesa".EstadoMesas[#Mesa].Rearme_CBx )
   END_RUNG wire#w2
   // the same network as SCL:
   "DB1_SalidasExterioresDeMesa".Mesa[#Mesa].Avanzar_E2E4 := ((((#PhsMx AND #PTF_Mx_MSig AND #NXT_Avance) OR NOT #PhsMx) AND NOT #Mem_CNT_Aus_salida AND #PosTR_S2 AND "DB902_Estado_ZonaMesa".EstadoMesas[#Mesa].Marcha_CBx AND NOT "DB900_Estado_Mesas".EstadoVI[#Mesa].Error_Mx) OR (NOT #Termico_S2 AND "DB902_Estado_ZonaMesa".EstadoMesas[#Mesa].Rearme_CBx)) AND #ok_tension;
END_REGION

REGION Network 8: Ir posicion 13
   // Dani Palacios: Prueba 16/04/2014
   RUNG wire#powerrail
      Contact( #Mem_CNT_Aus_salida )
      Contact( "DB902_Estado_ZonaMesa".EstadoMesas[#Mesa].Marcha_CBx )
      I_Contact( #PosTR_E1 )
      I_Contact( "DB900_Estado_Mesas".EstadoVI[#Mesa].Error_Mx )
      I_Contact( "DB902_Estado_ZonaMesa".EstadoMesas[#Mesa].ParoBlando_CBx )
      wire#w1
      Coil( "DB1_SalidasExterioresDeMesa".Mesa[#Mesa].Ir_Pos_E1E3 )
   END_RUNG
   RUNG wire#w1
      Coil( #TEMP_MA_TR_Pos_E1 )
   END_RUNG
   // the same network as SCL:
   #_w1 := #Mem_CNT_Aus_salida AND "DB902_Estado_ZonaMesa".EstadoMesas[#Mesa].Marcha_CBx AND NOT #PosTR_E1 AND NOT "DB900_Estado_Mesas".EstadoVI[#Mesa].Error_Mx AND NOT "DB902_Estado_ZonaMesa".EstadoMesas[#Mesa].ParoBlando_CBx;
   "DB1_SalidasExterioresDeMesa".Mesa[#Mesa].Ir_Pos_E1E3 := #Mem_CNT_Aus_salida AND "DB902_Estado_ZonaMesa".EstadoMesas[#Mesa].Marcha_CBx AND NOT #PosTR_E1 AND NOT "DB900_Estado_Mesas".EstadoVI[#Mesa].Error_Mx AND NOT "DB902_Estado_ZonaMesa".EstadoMesas[#Mesa].ParoBlando_CBx;
   #TEMP_MA_TR_Pos_E1 := #_w1;
END_REGION

REGION Network 9: ir posicion 24
   RUNG wire#powerrail
      Contact( #Mem_CNT_Pres_entrada )
      I_Contact( #Mem_CNT_Aus_salida )
      Contact( "DB902_Estado_ZonaMesa".EstadoMesas[#Mesa].Marcha_CBx )
      I_Contact( #PosTR_S2 )
      I_Contact( "DB900_Estado_Mesas".EstadoVI[#Mesa].Error_Mx )
      I_Contact( "DB902_Estado_ZonaMesa".EstadoMesas[#Mesa].ParoBlando_CBx )
      wire#w1
      Coil( "DB1_SalidasExterioresDeMesa".Mesa[#Mesa].Ir_Pos_E2E4 )
   END_RUNG
   RUNG wire#w1
      Coil( #TEMP_MA_TR_Pos_S2 )
   END_RUNG
   // the same network as SCL:
   #_w1 := #Mem_CNT_Pres_entrada AND NOT #Mem_CNT_Aus_salida AND "DB902_Estado_ZonaMesa".EstadoMesas[#Mesa].Marcha_CBx AND NOT #PosTR_S2 AND NOT "DB900_Estado_Mesas".EstadoVI[#Mesa].Error_Mx AND NOT "DB902_Estado_ZonaMesa".EstadoMesas[#Mesa].ParoBlando_CBx;
   "DB1_SalidasExterioresDeMesa".Mesa[#Mesa].Ir_Pos_E2E4 := #Mem_CNT_Pres_entrada AND NOT #Mem_CNT_Aus_salida AND "DB902_Estado_ZonaMesa".EstadoMesas[#Mesa].Marcha_CBx AND NOT #PosTR_S2 AND NOT "DB900_Estado_Mesas".EstadoVI[#Mesa].Error_Mx AND NOT "DB902_Estado_ZonaMesa".EstadoMesas[#Mesa].ParoBlando_CBx;
   #TEMP_MA_TR_Pos_S2 := #_w1;
END_REGION

REGION Network 10: nxt avtf
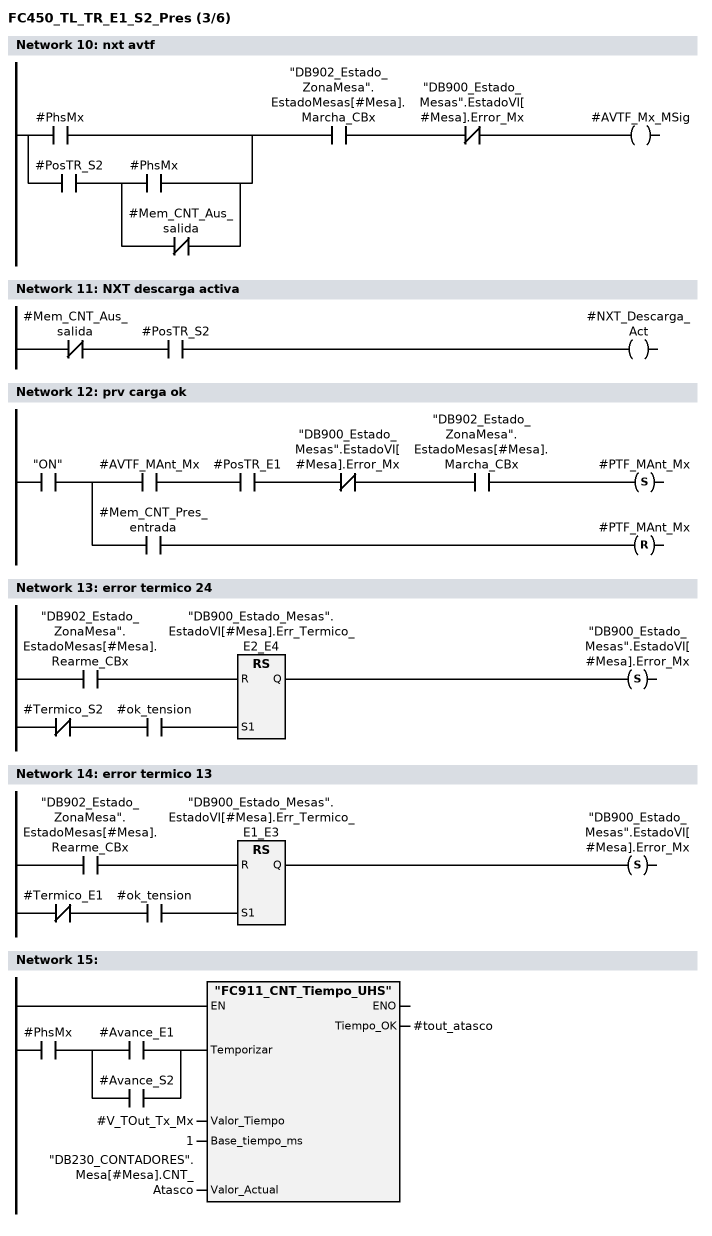
   RUNG wire#powerrail
      Contact( #PhsMx )
      wire#w1
      Contact( "DB902_Estado_ZonaMesa".EstadoMesas[#Mesa].Marcha_CBx )
      I_Contact( "DB900_Estado_Mesas".EstadoVI[#Mesa].Error_Mx )
      Coil( #AVTF_Mx_MSig )
   END_RUNG
   RUNG wire#powerrail
      Contact( #PosTR_S2 )
      wire#w2
      Contact( #PhsMx )
   END_RUNG wire#w1
   RUNG wire#w2
      I_Contact( #Mem_CNT_Aus_salida )
   END_RUNG wire#w1
   // the same network as SCL:
   #AVTF_Mx_MSig := (#PhsMx OR (#PosTR_S2 AND (#PhsMx OR NOT #Mem_CNT_Aus_salida))) AND "DB902_Estado_ZonaMesa".EstadoMesas[#Mesa].Marcha_CBx AND NOT "DB900_Estado_Mesas".EstadoVI[#Mesa].Error_Mx;
END_REGION

REGION Network 11: NXT descarga activa
   RUNG wire#powerrail
      I_Contact( #Mem_CNT_Aus_salida )
      Contact( #PosTR_S2 )
      Coil( #NXT_Descarga_Act )
   END_RUNG
   // the same network as SCL:
   #NXT_Descarga_Act := NOT #Mem_CNT_Aus_salida AND #PosTR_S2;
END_REGION

REGION Network 12: prv carga ok
   RUNG wire#powerrail
      Contact( "ON" )
      wire#w1
      Contact( #AVTF_MAnt_Mx )
      Contact( #PosTR_E1 )
      I_Contact( "DB900_Estado_Mesas".EstadoVI[#Mesa].Error_Mx )
      Contact( "DB902_Estado_ZonaMesa".EstadoMesas[#Mesa].Marcha_CBx )
      S_Coil( #PTF_MAnt_Mx )
   END_RUNG
   RUNG wire#w1
      Contact( #Mem_CNT_Pres_entrada )
      R_Coil( #PTF_MAnt_Mx )
   END_RUNG
   // the same network as SCL:
   IF "ON" AND #AVTF_MAnt_Mx AND #PosTR_E1 AND NOT "DB900_Estado_Mesas".EstadoVI[#Mesa].Error_Mx AND "DB902_Estado_ZonaMesa".EstadoMesas[#Mesa].Marcha_CBx THEN
       #PTF_MAnt_Mx := TRUE;
   END_IF;
   IF "ON" AND #Mem_CNT_Pres_entrada THEN #PTF_MAnt_Mx := FALSE; END_IF;
END_REGION

REGION Network 13: error termico 24
   RUNG wire#powerrail
      Contact( "DB902_Estado_ZonaMesa".EstadoMesas[#Mesa].Rearme_CBx )
      S_RS(operand := "DB900_Estado_Mesas".EstadoVI[#Mesa].Err_Termico_E2_E4, s1 := wire#w1)
      S_Coil( "DB900_Estado_Mesas".EstadoVI[#Mesa].Error_Mx )
   END_RUNG
   RUNG wire#powerrail
      I_Contact( #Termico_S2 )
      Contact( #ok_tension )
   END_RUNG wire#w1
   // the same network as SCL:
   IF "DB902_Estado_ZonaMesa".EstadoMesas[#Mesa].Rearme_CBx THEN
       "DB900_Estado_Mesas".EstadoVI[#Mesa].Err_Termico_E2_E4 := FALSE;   // RS flip-flop
   END_IF;
   IF NOT #Termico_S2 AND #ok_tension THEN
       "DB900_Estado_Mesas".EstadoVI[#Mesa].Err_Termico_E2_E4 := TRUE;
   END_IF;
   IF "DB900_Estado_Mesas".EstadoVI[#Mesa].Err_Termico_E2_E4 THEN
       "DB900_Estado_Mesas".EstadoVI[#Mesa].Error_Mx := TRUE;
   END_IF;
END_REGION

REGION Network 14: error termico 13
   RUNG wire#powerrail
      Contact( "DB902_Estado_ZonaMesa".EstadoMesas[#Mesa].Rearme_CBx )
      S_RS(operand := "DB900_Estado_Mesas".EstadoVI[#Mesa].Err_Termico_E1_E3, s1 := wire#w1)
      S_Coil( "DB900_Estado_Mesas".EstadoVI[#Mesa].Error_Mx )
   END_RUNG
   RUNG wire#powerrail
      I_Contact( #Termico_E1 )
      Contact( #ok_tension )
   END_RUNG wire#w1
   // the same network as SCL:
   IF "DB902_Estado_ZonaMesa".EstadoMesas[#Mesa].Rearme_CBx THEN
       "DB900_Estado_Mesas".EstadoVI[#Mesa].Err_Termico_E1_E3 := FALSE;   // RS flip-flop
   END_IF;
   IF NOT #Termico_E1 AND #ok_tension THEN
       "DB900_Estado_Mesas".EstadoVI[#Mesa].Err_Termico_E1_E3 := TRUE;
   END_IF;
   IF "DB900_Estado_Mesas".EstadoVI[#Mesa].Err_Termico_E1_E3 THEN
       "DB900_Estado_Mesas".EstadoVI[#Mesa].Error_Mx := TRUE;
   END_IF;
END_REGION

REGION Network 15
   RUNG wire#powerrail
      "FC911_CNT_Tiempo_UHS"(Temporizar := wire#w2, Valor_Tiempo := #V_TOut_Tx_Mx, Base_tiempo_ms := 1, Valor_Actual := "DB230_CONTADORES".Mesa[#Mesa].CNT_Atasco, Tiempo_OK => #tout_atasco)
   END_RUNG
   RUNG wire#powerrail
      Contact( #PhsMx )
      wire#w1
      Contact( #Avance_E1 )
   END_RUNG wire#w2
   RUNG wire#w1
      Contact( #Avance_S2 )
   END_RUNG wire#w2
   // the same network as SCL:
   "FC911_CNT_Tiempo_UHS"(Temporizar := #PhsMx AND (#Avance_E1 OR #Avance_S2),
                          Valor_Tiempo := #V_TOut_Tx_Mx,
                          Base_tiempo_ms := 1,
                          Valor_Actual := "DB230_CONTADORES".Mesa[#Mesa].CNT_Atasco,
                          Tiempo_OK => #tout_atasco);
END_REGION

REGION Network 16: Marca General Error
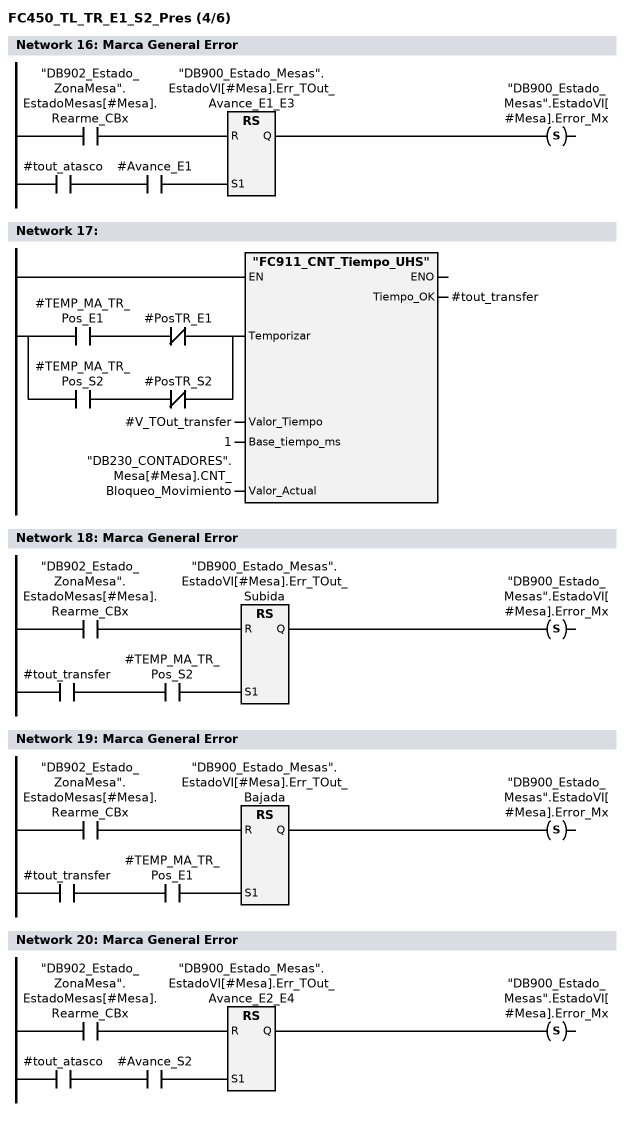
   RUNG wire#powerrail
      Contact( "DB902_Estado_ZonaMesa".EstadoMesas[#Mesa].Rearme_CBx )
      S_RS(operand := "DB900_Estado_Mesas".EstadoVI[#Mesa].Err_TOut_Avance_E1_E3, s1 := wire#w1)
      S_Coil( "DB900_Estado_Mesas".EstadoVI[#Mesa].Error_Mx )
   END_RUNG
   RUNG wire#powerrail
      Contact( #tout_atasco )
      Contact( #Avance_E1 )
   END_RUNG wire#w1
   // the same network as SCL:
   IF "DB902_Estado_ZonaMesa".EstadoMesas[#Mesa].Rearme_CBx THEN
       "DB900_Estado_Mesas".EstadoVI[#Mesa].Err_TOut_Avance_E1_E3 := FALSE;   // RS flip-flop
   END_IF;
   IF #tout_atasco AND #Avance_E1 THEN
       "DB900_Estado_Mesas".EstadoVI[#Mesa].Err_TOut_Avance_E1_E3 := TRUE;
   END_IF;
   IF "DB900_Estado_Mesas".EstadoVI[#Mesa].Err_TOut_Avance_E1_E3 THEN
       "DB900_Estado_Mesas".EstadoVI[#Mesa].Error_Mx := TRUE;
   END_IF;
END_REGION

REGION Network 17
   RUNG wire#powerrail
      "FC911_CNT_Tiempo_UHS"(Temporizar := wire#w1, Valor_Tiempo := #V_TOut_transfer, Base_tiempo_ms := 1, Valor_Actual := "DB230_CONTADORES".Mesa[#Mesa].CNT_Bloqueo_Movimiento, Tiempo_OK => #tout_transfer)
   END_RUNG
   RUNG wire#powerrail
      Contact( #TEMP_MA_TR_Pos_E1 )
      I_Contact( #PosTR_E1 )
   END_RUNG wire#w1
   RUNG wire#powerrail
      Contact( #TEMP_MA_TR_Pos_S2 )
      I_Contact( #PosTR_S2 )
   END_RUNG wire#w1
   // the same network as SCL:
   "FC911_CNT_Tiempo_UHS"(Temporizar := (#TEMP_MA_TR_Pos_E1 AND NOT #PosTR_E1) OR (#TEMP_MA_TR_Pos_S2 AND NOT #PosTR_S2),
                          Valor_Tiempo := #V_TOut_transfer,
                          Base_tiempo_ms := 1,
                          Valor_Actual := "DB230_CONTADORES".Mesa[#Mesa].CNT_Bloqueo_Movimiento,
                          Tiempo_OK => #tout_transfer);
END_REGION

REGION Network 18: Marca General Error
   RUNG wire#powerrail
      Contact( "DB902_Estado_ZonaMesa".EstadoMesas[#Mesa].Rearme_CBx )
      S_RS(operand := "DB900_Estado_Mesas".EstadoVI[#Mesa].Err_TOut_Subida, s1 := wire#w1)
      S_Coil( "DB900_Estado_Mesas".EstadoVI[#Mesa].Error_Mx )
   END_RUNG
   RUNG wire#powerrail
      Contact( #tout_transfer )
      Contact( #TEMP_MA_TR_Pos_S2 )
   END_RUNG wire#w1
   // the same network as SCL:
   IF "DB902_Estado_ZonaMesa".EstadoMesas[#Mesa].Rearme_CBx THEN
       "DB900_Estado_Mesas".EstadoVI[#Mesa].Err_TOut_Subida := FALSE;   // RS flip-flop
   END_IF;
   IF #tout_transfer AND #TEMP_MA_TR_Pos_S2 THEN
       "DB900_Estado_Mesas".EstadoVI[#Mesa].Err_TOut_Subida := TRUE;
   END_IF;
   IF "DB900_Estado_Mesas".EstadoVI[#Mesa].Err_TOut_Subida THEN
       "DB900_Estado_Mesas".EstadoVI[#Mesa].Error_Mx := TRUE;
   END_IF;
END_REGION

REGION Network 19: Marca General Error
   RUNG wire#powerrail
      Contact( "DB902_Estado_ZonaMesa".EstadoMesas[#Mesa].Rearme_CBx )
      S_RS(operand := "DB900_Estado_Mesas".EstadoVI[#Mesa].Err_TOut_Bajada, s1 := wire#w1)
      S_Coil( "DB900_Estado_Mesas".EstadoVI[#Mesa].Error_Mx )
   END_RUNG
   RUNG wire#powerrail
      Contact( #tout_transfer )
      Contact( #TEMP_MA_TR_Pos_E1 )
   END_RUNG wire#w1
   // the same network as SCL:
   IF "DB902_Estado_ZonaMesa".EstadoMesas[#Mesa].Rearme_CBx THEN
       "DB900_Estado_Mesas".EstadoVI[#Mesa].Err_TOut_Bajada := FALSE;   // RS flip-flop
   END_IF;
   IF #tout_transfer AND #TEMP_MA_TR_Pos_E1 THEN
       "DB900_Estado_Mesas".EstadoVI[#Mesa].Err_TOut_Bajada := TRUE;
   END_IF;
   IF "DB900_Estado_Mesas".EstadoVI[#Mesa].Err_TOut_Bajada THEN
       "DB900_Estado_Mesas".EstadoVI[#Mesa].Error_Mx := TRUE;
   END_IF;
END_REGION

REGION Network 20: Marca General Error
   RUNG wire#powerrail
      Contact( "DB902_Estado_ZonaMesa".EstadoMesas[#Mesa].Rearme_CBx )
      S_RS(operand := "DB900_Estado_Mesas".EstadoVI[#Mesa].Err_TOut_Avance_E2_E4, s1 := wire#w1)
      S_Coil( "DB900_Estado_Mesas".EstadoVI[#Mesa].Error_Mx )
   END_RUNG
   RUNG wire#powerrail
      Contact( #tout_atasco )
      Contact( #Avance_S2 )
   END_RUNG wire#w1
   // the same network as SCL:
   IF "DB902_Estado_ZonaMesa".EstadoMesas[#Mesa].Rearme_CBx THEN
       "DB900_Estado_Mesas".EstadoVI[#Mesa].Err_TOut_Avance_E2_E4 := FALSE;   // RS flip-flop
   END_IF;
   IF #tout_atasco AND #Avance_S2 THEN
       "DB900_Estado_Mesas".EstadoVI[#Mesa].Err_TOut_Avance_E2_E4 := TRUE;
   END_IF;
   IF "DB900_Estado_Mesas".EstadoVI[#Mesa].Err_TOut_Avance_E2_E4 THEN
       "DB900_Estado_Mesas".EstadoVI[#Mesa].Error_Mx := TRUE;
   END_IF;
END_REGION

REGION Network 21: Entradas Mesas
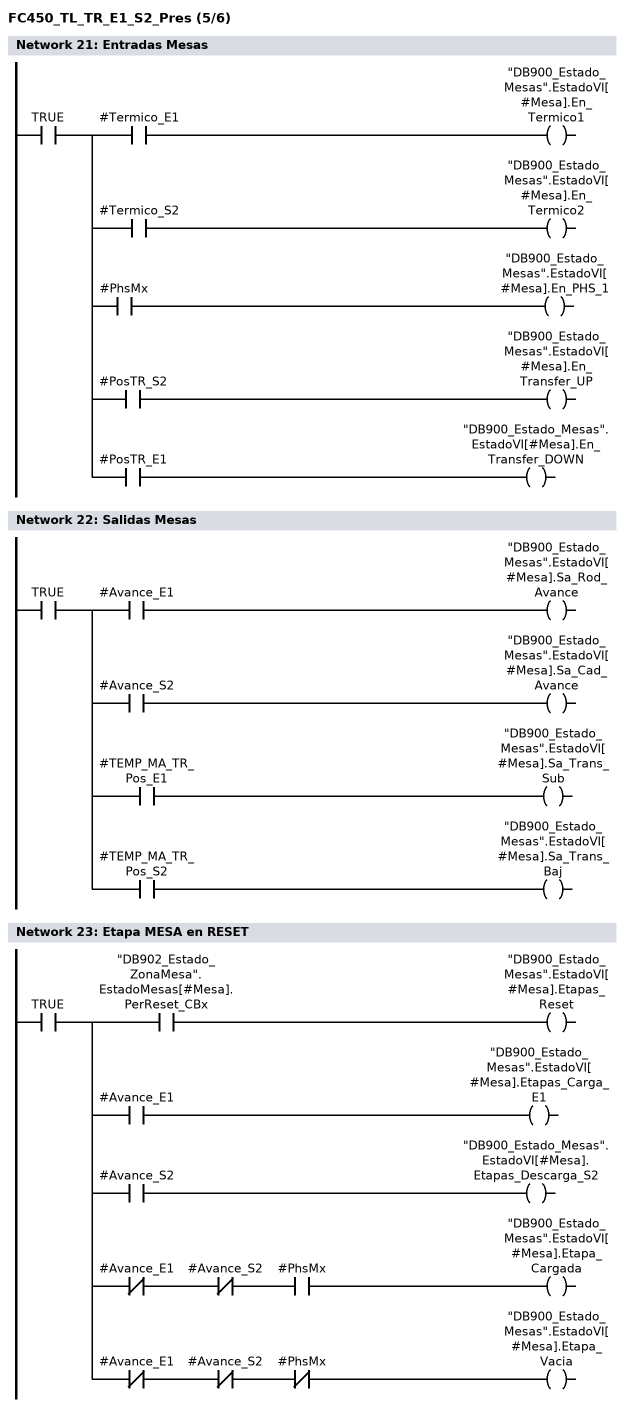
   RUNG wire#powerrail
      Contact( TRUE )
      wire#w1
      Contact( #Termico_E1 )
      Coil( "DB900_Estado_Mesas".EstadoVI[#Mesa].En_Termico1 )
   END_RUNG
   RUNG wire#w1
      Contact( #Termico_S2 )
      Coil( "DB900_Estado_Mesas".EstadoVI[#Mesa].En_Termico2 )
   END_RUNG
   RUNG wire#w1
      Contact( #PhsMx )
      Coil( "DB900_Estado_Mesas".EstadoVI[#Mesa].En_PHS_1 )
   END_RUNG
   RUNG wire#w1
      Contact( #PosTR_S2 )
      Coil( "DB900_Estado_Mesas".EstadoVI[#Mesa].En_Transfer_UP )
   END_RUNG
   RUNG wire#w1
      Contact( #PosTR_E1 )
      Coil( "DB900_Estado_Mesas".EstadoVI[#Mesa].En_Transfer_DOWN )
   END_RUNG
   // the same network as SCL:
   "DB900_Estado_Mesas".EstadoVI[#Mesa].En_Termico1 := TRUE AND #Termico_E1;
   "DB900_Estado_Mesas".EstadoVI[#Mesa].En_Termico2 := TRUE AND #Termico_S2;
   "DB900_Estado_Mesas".EstadoVI[#Mesa].En_PHS_1 := TRUE AND #PhsMx;
   "DB900_Estado_Mesas".EstadoVI[#Mesa].En_Transfer_UP := TRUE AND #PosTR_S2;
   "DB900_Estado_Mesas".EstadoVI[#Mesa].En_Transfer_DOWN := TRUE AND #PosTR_E1;
END_REGION

